  rx_DeleteMsgPart(pAnalyzeLastMessage := pAnalyzeLastMessage, nLen := nFindIndex , nPos := 1);
ELSE
  // end of message detected
  nFindIndex := FIND2(pAnalyzeLastMessage, ADR(');'));
  IF nFindIndex > 0 THEN
    (*Last sector is indicated with '-1'*)
    nSector := STRING_TO_DINT(LEFT(pAnalyzeLastMessage^, (UDINT_TO_INT(nFindIndex) - 1)));
  
    rx_DeleteMsgPart(pAnalyzeLastMessage := pAnalyzeLastMessage, nLen := nFindIndex + 1, nPos := 1);
  END_IF;
END_IF;

rx_ParseHeader := TRUE;
END_METHOD

(*
  Parse a point entry from string.
  And removes this string part from pAnalyzeLastMessage.
  :return: TRUE if point is valid
*)
METHOD PRIVATE rx_ParsePoint : BOOL
VAR_INPUT
  pAnalyzeLastMessage    : POINTER TO STRING(GVL_TcpIp.TCP_RXDATA_SIZE);  // telegram string for analysis
END_VAR
VAR_OUTPUT
  sCamResult             : ST_CameraPoint;
  bLast                  : BOOL;
END_VAR
VAR
  nFindIndex             : UDINT;
END_VAR
(*Index of mark (T)*)
nFindIndex := FIND2(pAnalyzeLastMessage, ADR(','));
IF nFindIndex > 0 THEN
  sCamResult.id := STRING_TO_UDINT(LEFT(pAnalyzeLastMessage^, (UDINT_TO_INT(nFindIndex) - 1)));
  
  rx_DeleteMsgPart(pAnalyzeLastMessage := pAnalyzeLastMessage, nLen := nFindIndex , nPos := 1);
END_IF;

(*rx*)
nFindIndex := FIND2(pAnalyzeLastMessage, ADR(','));
IF nFindIndex > 0 THEN
  sCamResult.x_ref := STRING_TO_DINT(LEFT(pAnalyzeLastMessage^, (UDINT_TO_INT(nFindIndex) - 1)));

  IF    (sCamResult.x_ref < cCameraMinXY)
     OR (sCamResult.x_ref > cCameraMaxXY)
  THEN
    sCamResult.valid := FALSE;
  END_IF;

  rx_DeleteMsgPart(pAnalyzeLastMessage := pAnalyzeLastMessage, nLen := nFindIndex , nPos := 1);
ELSE
  sCamResult.valid := FALSE;
END_IF;
(*ry*)
nFindIndex := FIND2(pAnalyzeLastMessage, ADR(','));
IF nFindIndex > 0 THEN
  sCamResult.y_ref := STRING_TO_DINT(LEFT(pAnalyzeLastMessage^, (UDINT_TO_INT(nFindIndex) - 1)));

  IF    (sCamResult.y_ref < cCameraMinXY)
     OR (sCamResult.y_ref > cCameraMaxXY)
  THEN
    sCamResult.valid := FALSE;
  END_IF;

  rx_DeleteMsgPart(pAnalyzeLastMessage := pAnalyzeLastMessage, nLen := nFindIndex , nPos := 1);
ELSE
  sCamResult.valid := FALSE;
END_IF;

(*lx*)
nFindIndex := FIND2(pAnalyzeLastMessage, ADR(','));
IF nFindIndex > 0 THEN
  sCamResult.lx := STRING_TO_DINT(LEFT(pAnalyzeLastMessage^, (UDINT_TO_INT(nFindIndex) - 1)));

  IF    (sCamResult.lx < cCameraMinXY)
     OR (sCamResult.lx > cCameraMaxXY)
  THEN
    sCamResult.valid := FALSE;
  END_IF;

  rx_DeleteMsgPart(pAnalyzeLastMessage := pAnalyzeLastMessage, nLen := nFindIndex , nPos := 1);
ELSE
  sCamResult.valid := FALSE;
END_IF;
(*ly*)
nFindIndex := FIND2(pAnalyzeLastMessage, ADR(','));
IF nFindIndex > 0 THEN
  sCamResult.ly := STRING_TO_DINT(LEFT(pAnalyzeLastMessage^, (UDINT_TO_INT(nFindIndex) - 1)));

  IF    (sCamResult.ly < cCameraMinXY)
     OR (sCamResult.ly > cCameraMaxXY)
  THEN
    sCamResult.valid := FALSE;
  END_IF;

  rx_DeleteMsgPart(pAnalyzeLastMessage := pAnalyzeLastMessage, nLen := nFindIndex , nPos := 1);
ELSE
  sCamResult.valid := FALSE;
END_IF;

(*v*)
nFindIndex := FIND2(pAnalyzeLastMessage, ADR(','));
IF nFindIndex > 0 THEN
  IF STRING_TO_INT(LEFT(pAnalyzeLastMessage^, (UDINT_TO_INT(nFindIndex) - 1))) = 1 THEN
    sCamResult.valid := TRUE;
  ELSE
    sCamResult.valid := FALSE;
  END_IF;

  rx_DeleteMsgPart(pAnalyzeLastMessage := pAnalyzeLastMessage, nLen := nFindIndex , nPos := 1);
ELSE
  sCamResult.valid := FALSE;
END_IF;
(*x*)
nFindIndex := FIND2(pAnalyzeLastMessage, ADR(','));
IF nFindIndex > 0 THEN
  sCamResult.x := STRING_TO_DINT(LEFT(pAnalyzeLastMessage^, (UDINT_TO_INT(nFindIndex) - 1)));

  IF    (sCamResult.x < cCameraMinXY)
     OR (sCamResult.x > cCameraMaxXY)
  THEN
    sCamResult.valid := FALSE;
  END_IF;

  rx_DeleteMsgPart(pAnalyzeLastMessage := pAnalyzeLastMessage, nLen := nFindIndex , nPos := 1);
ELSE
  sCamResult.valid := FALSE;
END_IF;
(*y*)
nFindIndex := FIND2(pAnalyzeLastMessage, ADR(','));
IF (nFindIndex > 0) AND (nFindIndex <= 8) THEN  (*nFindIndex is > 8 if a second message is in the frame*)
  sCamResult.y := STRING_TO_DINT(LEFT(pAnalyzeLastMessage^, (UDINT_TO_INT(nFindIndex) - 1)));

  IF    (sCamResult.y < cCameraMinXY)
     OR (sCamResult.y > cCameraMaxXY)
  THEN
    sCamResult.valid := FALSE;
  END_IF;

  rx_DeleteMsgPart(pAnalyzeLastMessage := pAnalyzeLastMessage, nLen := nFindIndex , nPos := 1);
ELSE
  nFindIndex := FIND2(pAnalyzeLastMessage, ADR(');'));
  IF nFindIndex > 0 THEN
    sCamResult.y := STRING_TO_DINT(LEFT(pAnalyzeLastMessage^, (UDINT_TO_INT(nFindIndex) - 1)));
    bLast := TRUE;
    IF    (sCamResult.y < cCameraMinXY)
       OR (sCamResult.y > cCameraMaxXY)
    THEN
      sCamResult.valid := FALSE;
    END_IF;

    rx_DeleteMsgPart(pAnalyzeLastMessage := pAnalyzeLastMessage, nLen := nFindIndex + 1, nPos := 1);
  ELSE
    sCamResult.valid := FALSE;
  END_IF;
END_IF;

rx_ParsePoint := sCamResult.valid;
END_METHOD

(*
  Parse rx test telegrams.
  :return: TRUE if it was a known test telegram, FALSE if other.
*)
METHOD PRIVATE rx_TestMsg : BOOL
VAR_INPUT
  pMessage    : POINTER TO STRING(GVL_TcpIp.TCP_RXDATA_SIZE);   // tcp message string pointer 
END_VAR
VAR
  nFIdx : UDINT;    // string find index
  nFrmIdx : UDINT;
  tDiff : LREAL;
  sTestMsg : T_MaxString;
END_VAR
// rx timestamp
_tTimeRx := F_GetCurDcTaskTime64();

// parse message type
nFIdx := FIND2(pMessage, ADR(sQvTest_Header));
IF nFIdx > 0 THEN  
  IF _bVerbose THEN
    LogLvl(Lvl:=E_LogSeverity.Debug, Msg:=F_Concat2('test_rx: msg received: ', pMessage^));
  END_IF
  
  // test telegram received
  DELETE2( pSrcString := pMessage
         , pDstString := ADR(sTestMsg)
         , nDstSize   := SIZEOF(sTestMsg)
         , nLen       := (nFIdx + INT_TO_UDINT(LEN(sQvTest_Header)) - 1)
         , nPos       := 1);

  // strip QR start and end characters
  FindAndDeleteChar(pSrcString:=ADR(sTestMsg), pDstString:=ADR(sTestMsg), nDstSize:=SIZEOF(sTestMsg), sDeleteChar:='<');
  FindAndDeleteChar(pSrcString:=ADR(sTestMsg), pDstString:=ADR(sTestMsg), nDstSize:=SIZEOF(sTestMsg), sDeleteChar:=';');
  
  // Parse per test message type, e.g.  <QR_CI_1;
  // -- qv input frame timing test
  IF sQvTest_CI = LEFT(sTestMsg, LEN(sQvTest_CI)) THEN
    // strip header and test indication
    DELETE2( pSrcString := ADR(sTestMsg)
           , pDstString := ADR(sTestMsg)
           , nDstSize   := SIZEOF(sTestMsg)
           , nLen       := (1 + INT_TO_UDINT(LEN(sQvTest_CI)) - 1)
           , nPos       := 1);
    // frame number
    nFrmIdx := TO_UINT(sTestMsg);
    IF nFrmIdx <= nC_MaxRxTimingEntries THEN
      _tTimeFrames_TestMsg[nFrmIdx] := F_GetCurDcTaskTime64();     // save test input frame timestamp
      _tTimeFramesMs_TestMsg[nFrmIdx] := TO_LREAL((_tTimeFrames_TestMsg[nFrmIdx]-_tTimeTrigger)/EC_DCTIME_TICKSPERMSEC64);
    END_IF
    rx_TestMsg := TRUE;
    
  // -- qv loop time test frame response
  ELSIF sQvTest_Loop = LEFT(sTestMsg, LEN(sQvTest_Loop)) THEN
    tDiff := TO_LREAL((_tTimeRx - _tTimeTx) / EC_DCTIME_TICKSPERMSEC64); // calc time elapsed in [ms]
    _sTimeElapsed := F_Concat2(TO_STRING(tDiff),'ms');
    LogLvl(Lvl:=E_LogSeverity.Debug, Msg:=F_Concat2('rx_test: Loop time=', _sTimeElapsed));
    rx_TestMsg := TRUE;
  
  // -- unknown test message
  ELSE
    ;
	END_IF
ELSE
  ; // other telegram
END_IF
END_METHOD

METHOD PRIVATE saveAuswertungPoint : ST_DeformationPointAccurate
VAR_INPUT
  sCamPoint : ST_CameraPoint;
END_VAR
VAR_OUTPUT
  bOK : BOOL;   // conversion has been done correctly (ok as well if point is invalid!)
END_VAR
VAR
  nMarkIndex        : UDINT;
  fDistortionFactor : LREAL;                 (*distortion factor*)
END_VAR
(*convert and save Auswertungs point*)
IF NOT getPointIndex(nId:=sCamPoint.id, nIndex=>nMarkIndex) THEN
  LogError(F_Concat3('Auswertung point with Id: ', TO_STRING(sCamPoint.id), ' not found, ignore'));
  bOK := FALSE;
  RETURN;
END_IF

(*----- calculate print point position -----*)
(*Actual position of distinctive mark*)
(*NOTE: camera points have a different resolution! camera 300dpi * 16=4800dpi*)
IF sTeachPoints[nMarkIndex].x_teach_Print = 0 THEN 
  (*Fully automatic mode*)
  sTeachPoints[nMarkIndex].x_Print := FC_CONV_SUBPX_TO_M( sCamPoint.y
                                                          , LREAL_TO_UDINT(cCameraResolution)
                                                          , LREAL_TO_UDINT(cCameraResolutionSubpixel)) * 1000;  (*[m] => [mm]*)
ELSE
  (*Semi automatic mode*)
  sTeachPoints[nMarkIndex].x_Print :=     sTeachPoints[nMarkIndex].x_ref_Print
                                        + sTeachPoints[nMarkIndex].x_teach_Print
                                        - FC_CONV_SUBPX_TO_M( sCamPoint.y
                                                            , LREAL_TO_UDINT(cCameraResolution)
                                                            , LREAL_TO_UDINT(cCameraResolutionSubpixel)) * 1000;  (*[m] => [mm]*)
END_IF;
IF sTeachPoints[nMarkIndex].y_teach_Print = 0 THEN 
  (*Fully automatic mode*)
  sTeachPoints[nMarkIndex].y_Print :=   ((fPrintUnitWidthTAct/2 + fCameraWidthTC/2) * 1000)  (*[m] => [mm]*)
                                        - (  DINT_TO_LREAL(sCamPoint.x)
                                           / (fCameraRealResolution * cCameraResolutionSubpixel) * 25.4);  (*[mm]*)
ELSE
  (*Semi automatic mode*)
  sTeachPoints[nMarkIndex].y_Print :=     sTeachPoints[nMarkIndex].y_ref_Print
                                        + sTeachPoints[nMarkIndex].y_teach_Print
                                        - (  DINT_TO_LREAL(sCamPoint.x)
                                           / (fCameraRealResolution * cCameraResolutionSubpixel) * 25.4);  (*[mm]*)
END_IF;

// save cam point for visu
sCameraPoints[nMarkIndex] := sCamPoint;

(*----- create cam correction point -----*)
(*NOTE: correction will be rounded to [px]*)
saveAuswertungPoint.x_ref := F_MeterToSubPixelReal( sTeachPoints[nMarkIndex].x_ref_Print * 0.001      (*[mm] => [m]*)
                                     , UDINT_TO_LREAL(_nPrintUnitResolution));             (*Result should be in pixels*)                           
saveAuswertungPoint.y_ref := F_MeterToSubPixelReal( sTeachPoints[nMarkIndex].y_ref_Print * 0.001      (*[mm] => [m]*)
                                     , UDINT_TO_LREAL(_nPrintUnitResolution));             (*Result should be in pixels*)       
fCameraDelay := F_SubPixelToMeter(lPosSubPx:=_nCamStartPosDeviation, fResSubPx:=UDINT_TO_LREAL(_nPrintUnitResolution*_nPrintUnitSubPx));
saveAuswertungPoint.dx    := F_MeterToSubPixelReal( (sTeachPoints[nMarkIndex].x_ref_Print - sTeachPoints[nMarkIndex].x_Print) * 0.001  (*[mm] => [m]*)
                                     + fCameraDelay                                        (*apply camera trigger jitter*)
                                     , UDINT_TO_LREAL(_nPrintUnitResolution));             (*Result should be in pixels*)
                                     
(*Distortion due to expansion of print unit, calculate factor*)
fDistortionFactor := ((_fPrintUnitWidthTC / 2 * 1000) - sTeachPoints[nMarkIndex].y_ref_Print) / (_fPrintUnitWidthTC / 2 * 1000);
saveAuswertungPoint.dy := F_MeterToSubPixelReal( (  (sTeachPoints[nMarkIndex].y_ref_Print - sTeachPoints[nMarkIndex].y_Print)
                                     + fCameraAdjustmentY
                                     + ((fPrintUnitWidthDiff * 1000 / 2) * fDistortionFactor)   (*Distortion due to expansion of print unit*)
                                     + (fPrintUnitCenterOffsetTAct - fCameraCenterOffsetTAct)   (*Compensation due to unilateral expansion*)
                                    ) * 0.001  (*[mm] => [m]*)
                                  , UDINT_TO_LREAL(_nPrintUnitResolution));             (*Result should be in pixels*)
                                  
// not used entries
saveAuswertungPoint.index := 0; // optional: TO_DINT(sCamPoint.id);
saveAuswertungPoint.col := 0;
saveAuswertungPoint.row := 0;
saveAuswertungPoint.valid := sCamPoint.valid;
IF NOT sCamPoint.valid THEN     // erase spurious corrections on invalid points
  saveAuswertungPoint.dx := 0;
  saveAuswertungPoint.dy := 0;
END_IF
nNbMarksScanned := nNbMarksScanned + 1;
bOK := TRUE;
END_METHOD

METHOD PRIVATE saveTeachPoint
VAR_INPUT
  sCamPoint : ST_CameraPoint;
END_VAR
(*save teach point in table*)
// NOTE: mark ID unique and does not match the array index! 
IF nNbMarksTeach = GVL_Camera.cMaxNbMarks THEN 
  LogLvl(Lvl:=E_LogSeverity.Error, Msg:=F_Concat4('Too many marks received max. allowed: ', TO_STRING(GVL_Camera.cMaxNbMarks), ' ignore mark with id:', TO_STRING(sCamPoint.id)));
  RETURN;
END_IF

// save next teach mark
nNbMarksTeach := nNbMarksTeach + 1;
sCameraPoints[nNbMarksTeach] := sCamPoint;
END_METHOD

(*
  Set mode to camera.
  :return: TRUE if success
*)
METHOD setCameraMode : BOOL
VAR_INPUT
  eCameraMode : E_CameraMode;
END_VAR
IF eCameraMode = E_CameraMode.XYR OR   // supported modi
   eCameraMode = E_CameraMode.Auto OR
   eCameraMode = E_CameraMode.Live OR 
   eCameraMode = E_CameraMode.Trend THEN
   
  _eCameraMode := eCameraMode;  // set desired mode
  setCameraMode := TRUE;
ELSE
  LogError(F_Concat3('Camera mode=', TO_STRING(eCameraMode), ' not supported by camera'));
  _eCameraMode := E_CameraMode.NoCorrection;
END_IF
END_METHOD

METHOD SimEnter : BOOL
VAR_INST
  sSimMsg         : CalmarCompTcpIp.ST_TcpMsg;
  nFrameSize      : UDINT := 2048;
  nMarksPerFrame  : UDINT := 4;
END_VAR
IF NOT bSimEnable THEN RETURN; END_IF

IF    _nSimMode = 0 THEN
   //nNbMarksTeach := 4; // just somebigger than 2
   //nNbMarks := nNbMarksTeach;
ELSIF _nSimMode = 1 THEN
  // use external camera simulation script
  nFrameNr := 0;
ELSIF _nSimMode = 2 THEN
  // send directly some messages
  sSimMsg.stRemoteAddr.sAddr:='127.0.0.1';
  sSimMsg.stRemoteAddr.nPort:=3000;
  //v100 teach
  //rx_callback(sMessage:='<position(100,T,39,3,125,0,0,0,0,1,7184,7184,126,0,0,0,0,1,7184,26080,127,0,0,0,0,1,7184,35520,128,0,0,0,0,1,7184,54416,129,0,0,0,0,1,7168,73312,130,0,0,0,0,1,7184,82768,131,0,0,0,0,1,7184,101664,132,0,0,0,0,1,7184,120560,133,0,0,0,0,1,7184,139456,134,0,0,0,0,1,7184,148912,135,0,0,0,0,1,7184,167808,136,0,0,0,0,1,7168,186704,137,0,0,0,0,1,63872,7184,138,0,0,0,0,1,63872,26080,139,0,0,0,0,1,63872,35520,140,0,0,0,0,1,63872,54416,141,0,0,0,0,1,63872,73312,142,0,0,0,0,1,63872,82768,143,0,0,0,0,1,63872,101664,144,0,0,0,0,1,63872,120560,145,0,0,0,0,1,63872,139456,146,0,0,0,0,1,63872,148912,147,0,0,0,0,1,63872,167808,148,0,0,0,0,1,63872,186704,149,0,0,0,0,1,130016,7168,150,0,0,0,0,1,130016,26080,151,0,0,0,0,1,130016,35520,152,0,0,0,0,1,130016,54416,153,0,0,0,0,1,130016,73312,154,0,0,0,0,1,130016,82768,155,0,0,0,0,1,130016,101664,156,0,0,0,0,1,130016,120560,157,0,0,0,0,1,130016,139456,158,0,0,0,0,1,130016,148912,159,0,0,0,0,1,130016,167808,160,0,0,0,0,1,130016,186704,161,0,0,0,0,1,35520,7168,162,0,0,0,0,1,35520,5441);');
  //v110 teach
  sSimMsg.sMessage:= '<position(110,T,38,12,1,0,0,0,0,1,7184,7184,2,0,0,0,0,1,7184,26080,4,0,0,0,0,1,7184,35520,128,0,0,0,0,1,7184,54416,5,0,0,0,0,1,7168,73312,130,0,0,0,0,1,7184,82768,131,0,0,0,0,1,7184,101664,132,0,0,0,0,1,7184,120560,133,0,0,0,0,1,7184,139456,134,0,0,0,0,1,7184,148912,135,0,0,0,0,1,7184,167808,136,0,0,0,0,1,7168,186704,137,0,0,0,0,1,63872,7184,138,0,0,0,0,1,63872,26080,139,0,0,0,0,1,63872,35520,140,0,0,0,0,1,63872,54416,141,0,0,0,0,1,63872,73312,142,0,0,0,0,1,63872,82768,143,0,0,0,0,1,63872,101664,144,0,0,0,0,1,63872,120560,145,0,0,0,0,1,63872,139456,146,0,0,0,0,1,63872,148912,147,0,0,0,0,1,63872,167808,148,0,0,0,0,1,63872,186704,149,0,0,0,0,1,130016,7168,150,0,0,0,0,1,130016,26080,151,0,0,0,0,1,130016,35520,152,0,0,0,0,1,130016,54416,153,0,0,0,0,1,130016,73312,154,0,0,0,0,1,130016,82768,155,0,0,0,0,1,130016,101664,156,0,0,0,0,1,130016,120560,157,0,0,0,0,1,130016,139456,158,0,0,0,0,1,130016,148912,159,0,0,0,0,1,130016,167808,160,0,0,0,0,1,130016,186704,161,0,0,0,0,1,35520,7168,162,0,0,0,0,1,35520,5441);';
  //points 1 to 38
  //sSimMsg.sMessage:= '<position(110,T,38,12,1,0,0,0,0,1,7184,7184,2,0,0,0,0,1,7184,26080,3,0,0,0,0,1,7184,35520,4,0,0,0,0,1,7184,54416,5,0,0,0,0,1,7168,73312,6,0,0,0,0,1,7184,82768,7,0,0,0,0,1,7184,101664,8,0,0,0,0,1,7184,120560,9,0,0,0,0,1,7184,139456,10,0,0,0,0,1,7184,148912,11,0,0,0,0,1,7184,167808,12,0,0,0,0,1,7168,186704,13,0,0,0,0,1,63872,7184,14,0,0,0,0,1,63872,26080,15,0,0,0,0,1,63872,35520,16,0,0,0,0,1,63872,54416,17,0,0,0,0,1,63872,73312,18,0,0,0,0,1,63872,82768,19,0,0,0,0,1,63872,101664,20,0,0,0,0,1,63872,120560,21,0,0,0,0,1,63872,139456,22,0,0,0,0,1,63872,148912,23,0,0,0,0,1,63872,167808,24,0,0,0,0,1,63872,186704,25,0,0,0,0,1,130016,7168,26,0,0,0,0,1,130016,26080,27,0,0,0,0,1,130016,35520,28,0,0,0,0,1,130016,54416,29,0,0,0,0,1,130016,73312,30,0,0,0,0,1,130016,82768,31,0,0,0,0,1,130016,101664,32,0,0,0,0,1,130016,120560,33,0,0,0,0,1,130016,139456,34,0,0,0,0,1,130016,148912,35,0,0,0,0,1,130016,167808,36,0,0,0,0,1,130016,186704,37,0,0,0,0,1,35520,7168,38,0,0,0,0,1,35520,5441);';
  rx_callback(sMessage:=sSimMsg);
END_IF
END_METHOD

METHOD SimExit : BOOL
IF NOT bSimEnable THEN RETURN; END_IF

IF    _nSimMode = 0 THEN
  ;  // no action
ELSIF _nSimMode = 1 THEN
  nFrameNr := 0;
ELSIF _nSimMode = 2 THEN
  ;  // no action
END_IF
END_METHOD

(*
  External camera simulation script. 
  Simulates the line camera. Opens a TcpIp server where the the linecam plc client can conect to...
*)
METHOD SimulateCamera
VAR_INST
  rfTrig_En : RF_TRIG;
  tOnFrame  : TON;
END_VAR
VAR
  ams_host : STRING;
  ams_port : UINT;
  cmd : STRING;
  
  tFrameTime : TIME;
END_VAR
IF _nSimMode <> 1 THEN RETURN; END_IF   // only cam simulation

// simulation enable / disable
rfTrig_En(CLK:=_bSimulate);
IF rfTrig_En.RT THEN 
  // --- start simulation -----
  LogLvl(Lvl:=E_LogSeverity.Debug, Msg:='Start CamSimulation');

  fbScriptCamSim.Init(sScriptDir:=F_Concat2(_aCamSimScriptPath, 'Tools\CameraTest\'));
  fbScriptCamSim.sStartScriptName := 'Start.bat';
  (* Script parameter:
    parser.add_argument("ams_host", help="AmsNetId of host system")
    parser.add_argument("ams_port", help="AmsPort of host system", type=int)
    parser.add_argument("plc_path", help="plc interface (base) path")
    parser.add_argument("cam_ip", help="camera ip address")
    parser.add_argument("cam_port", help="camera port")
    parser.add_argument("--sim_mode", help="simulation enabled", type=bool)
  *)
  // build cmd line string dynamically 
  ams_host := '';
  ams_port := TwinCAT_SystemInfoVarList._AppInfo.AdsPort; 
  cmd := F_Concat7(ams_host,' ',TO_STRING(ams_port),' ',THIS^.InstanceName,' ',F_Concat3('127.0.0.1',' ',TO_STRING(5030)));
  fbScriptCamSim.Start(cmd);
  
ELSIF rfTrig_En.FT THEN 
  // --- stop/exit simulation ------
  LogLvl(Lvl:=E_LogSeverity.Debug, Msg:='Stop CamSimulation');
  // stop script
  fbScriptCamSim.Stop(nPID := THIS^.nScriptPID);
END_IF

// --- run script command ------
IF NOT fbScriptCamSim.bBusy THEN 
  IF fbScriptCamSim.bError THEN //Launch error
    LogError(F_Concat2('Script error=', TO_STRING(fbScriptCamSim.nErrId)));
  ELSE //Launch done
    ;
  END_IF
END_IF

// --- script live interface -------
IF _bCamTriggerStarted THEN
  IF tOnFrame.Q THEN
    nFrameNr := nFrameNr + 1; // demand next frame
	END_IF
  tFrameTime := REAL_TO_TIME(((84.6667 / 1_000_000) * 0.5)*1000*1024);  // 1024px @300dpi with speed 0.5m/s
  tOnFrame(IN:=NOT tOnFrame.Q, PT:=tFrameTime);
END_IF
END_METHOD

METHOD SimUpdate : BOOL
VAR_INST
  rfTrigCamTrigger : RF_TRIG;
  sSimMsg          : CalmarCompTcpIp.ST_TcpMsg;
END_VAR
// simulation handling
_rfTrigSim(CLK:=_bSimulate);
IF _rfTrigSim.RT THEN    SimEnter();
ELSIF _rfTrigSim.FT THEN SimExit(); END_IF
IF NOT _bSimulate THEN RETURN; END_IF

// we are in simulation mode
// - triggered
rfTrigCamTrigger(CLK:=_bCamTriggerStarted);

IF    _nSimMode = 0 THEN
  // direct points stream of all points in trigger
  IF rfTrigCamTrigger.RT THEN
     CreateSimCamPoints();
     _ePossibleMode := E_CameraMode.Live;
  END_IF
  // stream points
  StreamSimCamPoint();
 
ELSIF _nSimMode = 1 THEN
  // use external camera simulation script
  SimulateCamera();
  
ELSIF _nSimMode = 2 THEN
  IF rfTrigCamTrigger.RT THEN
    // send directly some messages
    sSimMsg.sMessage:='<position(110,A,5,1,125,0,0,0,0,1,12196,9766,137,0,0,0,0,1,69013,9660,149,0,0,0,0,1,135374,9496,161,0,0,0,0,1,40589,9699,163,0,0,0,0,1,116414,9527);';
    rx_callback(sMessage:=sSimMsg);
    sSimMsg.sMessage:='<position(110,A,3,2,126,0,0,0,0,1,11602,28300,138,0,0,0,0,1,68917,28190,150,0,0,0,0,1,136214,27951);';
    // also posible: sSimMsg.sMessage:='<position(110,A,3,2,126,0,0,0,0,1,11602,28300,138,0,0,0,0,1,68917,28190,150,0,0,0,0,1,136214,27951);<position(110,A,0,-1);';
    rx_callback(sMessage:=sSimMsg);
    sSimMsg.sMessage:='<position(110,A,0,-1);';
    rx_callback(sMessage:=sSimMsg);
  END_IF
END_IF


tx_test();
END_METHOD

{attribute 'monitoring':='variable'}
PROPERTY sName : STRING
GET
sName := 'LineCam Base';
END_GET
END_PROPERTY

(*
  Sort sCameraPoints list with ascending [.id] 
*)
METHOD sortPoints
VAR
  i, k : UDINT;
  tmpPoint : ST_CameraPoint;
END_VAR
// sort array (increasing id)
FOR i := 1 TO nNbMarksTeach DO
  FOR k := 1 TO nNbMarksTeach-1 DO
    IF sCameraPoints[k].id > sCameraPoints[k+1].id THEN
      tmpPoint := sCameraPoints[k+1];
      sCameraPoints[k+1] := sCameraPoints[k];
      sCameraPoints[k] := tmpPoint;
    END_IF
	END_FOR
END_FOR
END_METHOD

METHOD PRIVATE StreamSimCamPoint : BOOL
VAR_INPUT
END_VAR
VAR
 tCurrent : T_DCTIME64;
 tElapsed : LREAL;
 tCol : LREAL;
 nCol : UDINT;
 nPointCt : UDINT;
 tFrameFirstDelayFix : LREAL := 50; // deleat to first received frame after trigger
 tFrameTimeJitterMax : LREAL := 30; // max. process time for a camera frame to be received after a simulated scan [ms]
END_VAR
VAR_INST
 fbRand : DRAND;
END_VAR
IF IfSpeed = 0 THEN RETURN; END_IF

fbRand();
tCurrent := F_GetCurDcTaskTime64();             // current time 
tElapsed := TO_LREAL((tCurrent-_tTimeTrigger)   // time elapsed after trigger
                  / EC_DCTIME_TICKSPERMSEC64); 
tCol := F_SubPixelToMeter(                      // time for one column  in [ms] 
                  lPosSubPx:=TO_DINT(_nSimCamFrameDepth), 
                  fResSubPx:=_nPrintUnitResolution) * 1000 / IfSpeed;
tElapsed := tElapsed-tFrameFirstDelayFix-(tFrameTimeJitterMax * fbRand.Num);
IF tElapsed < 0 THEN nCol := 0;
ELSE                 nCol := TO_UDINT(tElapsed / tCol);  // current column number
END_IF

nPointCt := nCol*_nSimCamMarksPerFrame;         // current number of points to be streamed

// stream new points
WHILE nNbMarksScanned < nPointCt AND nNbMarksScanned < nNbMarks DO
  // add to container
  IF _iCameraSink<>0 THEN
    stCamPoint := _sSimCamPoints[nNbMarksScanned+1];
    _iCameraSink.AddCamPoint(stCamPoint);
    // add scanned marks
  END_IF;
  nNbMarksScanned := nNbMarksScanned + 1;
END_WHILE
END_METHOD

METHOD PRIVATE tx_test : BOOL
VAR_INPUT
END_VAR
VAR_INST
  _sTestTxMsg               : T_MaxString;
END_VAR
IF _pFbTcpIpClient = 0 THEN RETURN; END_IF

// sent a test message to QR
IF _bTestTx THEN
  _sTestTxMsg := F_Concat4('<', sQvTest_Header, sQvTest_Loop, ';');
  _tTimeTx := F_GetCurDcTaskTime64();
  _pFbTcpIpClient^.send(sMessage:=_sTestTxMsg);
  LogLvl(Lvl:=E_LogSeverity.Debug, Msg:=F_Concat2('test_tx sent: ', _sTestTxMsg));
  _bTestTx := FALSE;
END_IF
END_METHOD

(*
  Check teach points for validy and quality.
*)
METHOD verifyTeachPoints : BOOL
VAR
  lCtr : UDINT;
END_VAR

IF _fFrameLength <> 0 THEN
  nNumFrames := LIMIT(1, TO_UDINT(FC_LREAL_TO_DINT((fImageLength / _fFrameLength) + 1)), GVL_Camera.cMaxNbSectors); 
END_IF
bNotAllFramesContainTeachPoints := FALSE;
FOR lCtr := 1 TO nNumFrames DO
  IF nNumPointsPerSectorT[lCtr] = 0 THEN
    bNotAllFramesContainTeachPoints := TRUE;
	END_IF
END_FOR


bNotEnoughTeachPoints := FALSE;
IF    nNumPointsPerSectorT[1] < 2  THEN _ePossibleMode := E_CameraMode.NoCorrection; bNotEnoughTeachPoints := TRUE; //< 2 points in first frame
ELSIF nNumPointsPerSectorT[1] <= 2 THEN _ePossibleMode := E_CameraMode.XYR;          bNotEnoughTeachPoints := TRUE; //< 3 points in first frame
ELSE
  _ePossibleMode := E_CameraMode.Live;
END_IF


// teach is valid
_bTeachOk       := TRUE;
END_METHOD

END_FUNCTION_BLOCK

// ---- POUs/Print/Camera/LineCamera/FB_LineCamera106.TcPOU
(*
  QualiVision line camera system
  DMAX106.   
*)
FUNCTION_BLOCK FB_LineCamera106 EXTENDS FB_LineCamera

VAR CONSTANT
  cCameraWidth106           : DINT := 13440;   (*Camera width [px]*)
  cCameraMechOffsetTC106    : REAL :=  88.0;   (*Camera mechanical offset at calibration temp [mm]*)
  cMechOffsetCameraToPU106  : REAL :=  30.31;  (*Camera mechanical offset to PrintUnit [mm]*)
  cPrintUnitMechOffsetTC106 : REAL := 31.4747; (*PrintUnit mechanical offset at calibration temp [mm]*)
END_VAR

SUPER^();

METHOD InitLineCamera
VAR_INPUT
  nPrintUnitResolution         : UDINT;    (*printhead pixel resolution [dpi]*)
  nPrintUnitSubPx              : UDINT;    (*print unit subPixel resolution [SubPx]*)
  nPrintUnitWidth              : UDINT;    (*print unit width in [px]*)
  iCameraTrigger               : I_CameraTrigger;
END_VAR
(*Init for dmax type*)
_nCameraWidth           := cCameraWidth106;
_fCameraMechOffsetTC    := cCameraMechOffsetTC106;
_fMechOffsetCameraToPU  := cMechOffsetCameraToPU106;
_fPrintUnitMechOffsetTC := cPrintUnitMechOffsetTC106;

SUPER^.InitLineCamera( nPrintUnitResolution := nPrintUnitResolution
                      , nPrintUnitSubPx := nPrintUnitSubPx
                      , nPrintUnitWidth := nPrintUnitWidth
                      , iCameraTrigger := iCameraTrigger);
END_METHOD

{attribute 'monitoring':='variable'}
PROPERTY sName : STRING
GET
sName := 'LineCam 106';
END_GET
END_PROPERTY

END_FUNCTION_BLOCK

// ---- POUs/Print/Camera/LineCamera/FB_LineCamera76.TcPOU
(*
  QualiVision line camera system
  DMAX76.   
*)
FUNCTION_BLOCK FB_LineCamera76 EXTENDS FB_LineCamera

VAR CONSTANT
  cCameraWidth76            : DINT :=  9216;   (*Camera width [px]*)
  cCameraMechOffsetTC76     : REAL := 101.5;   (*Camera mechanical offset at calibration temp [mm]*)
  cMechOffsetCameraToPU76   : REAL :=  13.039; (*Camera mechanical offset to PrintUnit [mm]*)
  cPrintUnitMechOffsetTC76  : REAL := 32.9869; (*PrintUnit mechanical offset at calibration temp [mm]*)
END_VAR

SUPER^();

METHOD InitLineCamera
VAR_INPUT
  nPrintUnitResolution         : UDINT;    (*printhead pixel resolution [dpi]*)
  nPrintUnitSubPx              : UDINT;    (*print unit subPixel resolution [SubPx]*)
  nPrintUnitWidth              : UDINT;    (*print unit width in [px]*)
  iCameraTrigger               : I_CameraTrigger;
END_VAR
(*Init for dmax type*)
_nCameraWidth           := cCameraWidth76;
_fCameraMechOffsetTC    := cCameraMechOffsetTC76;
_fMechOffsetCameraToPU  := cMechOffsetCameraToPU76;
_fPrintUnitMechOffsetTC := cPrintUnitMechOffsetTC76;

SUPER^.InitLineCamera( nPrintUnitResolution := nPrintUnitResolution
                      , nPrintUnitSubPx := nPrintUnitSubPx
                      , nPrintUnitWidth := nPrintUnitWidth
                      , iCameraTrigger := iCameraTrigger);
END_METHOD

{attribute 'monitoring':='variable'}
PROPERTY sName : STRING
GET
sName := 'LineCam 76';
END_GET
END_PROPERTY

END_FUNCTION_BLOCK

// ---- POUs/Print/Camera/LineCamera/FB_LineCamera585.TcPOU
(*
  QualiVision line camera system
  DMAX76.   
*)
FUNCTION_BLOCK FB_LineCamera585 EXTENDS FB_LineCamera

VAR CONSTANT
  cCameraWidth585            : DINT := 9216;     (*Camera width [px]*)
  cCameraMechOffsetTC585     : REAL := 101.5;    (*Camera mechanical offset at calibration temp [mm]*)
  cMechOffsetCameraToPU585   : REAL :=  13.039;  (*Camera mechanical offset to PrintUnit [mm]*)
  cPrintUnitMechOffsetTC585  : REAL :=  32.9869; (*PrintUnit mechanical offset at calibration temp [mm]*)
END_VAR

SUPER^();

METHOD InitLineCamera
VAR_INPUT
  nPrintUnitResolution         : UDINT;    (*printhead pixel resolution [dpi]*)
  nPrintUnitSubPx              : UDINT;    (*print unit subPixel resolution [SubPx]*)
  nPrintUnitWidth              : UDINT;    (*print unit width in [px]*)
  iCameraTrigger               : I_CameraTrigger;
END_VAR
(*Init for dmax type*)
_nCameraWidth           := cCameraWidth585;
_fCameraMechOffsetTC    := cCameraMechOffsetTC585;
_fMechOffsetCameraToPU  := cMechOffsetCameraToPU585;
_fPrintUnitMechOffsetTC := cPrintUnitMechOffsetTC585;

SUPER^.InitLineCamera( nPrintUnitResolution := nPrintUnitResolution
                     , nPrintUnitSubPx      := nPrintUnitSubPx
                     , nPrintUnitWidth      := nPrintUnitWidth
                     , iCameraTrigger       := iCameraTrigger
                     );
END_METHOD

{attribute 'monitoring':='variable'}
PROPERTY sName : STRING
GET
sName := 'LineCam 585';
END_GET
END_PROPERTY

END_FUNCTION_BLOCK

// ---- POUs/Print/Camera/MarkCameraWEU/FB_MarkCamera_WEU.TcPOU
(*
  Mark camera system on WEU machine
  1 mark sensor (optional: reverse mode - roll printed in reversed direction, sensor moved to other side)
*)
FUNCTION_BLOCK FB_MarkCamera_WEU EXTENDS FB_CameraBase
VAR_INPUT
  bReadyForPrinting             : BOOL;     // 
  nCurrentPosition              : DINT;     // current print postion
  fCurrentSpeed                 : LREAL;    // current print speed
  bPrintMarkExist               : BOOL;     // [from machine] print mark existing
  bPrintDirReverse              : BOOL;     // [from machine] print substrate in reverse direction
  nUsePerRepeatInLine           : UDINT;    // [from machine] use per repeat
  fMarkSizeDefault              : LREAL;    // mark size "a" [m]
  fMarkDistRepeatToStartMark    : LREAL;    // mark distance from repeat to start mark [m]
  fMarkDistFromCenter           : LREAL;    // mark distance from center [m]
END_VAR
VAR
  fbMarkDefinition   : FB_MarkDefinition;   // mark definition instance (used by MarkDetection)
  fbMarkDetection    : FB_MarkDetection;    // StartPosTrigger, CameraTrigger and MarkDetection (Mark handler for MarkCamera)
  
  // teach info
  _bTeachOk                     : BOOL;
  _nTeachedPoints               : UDINT;
  _nDetectedMarks               : UDINT;
  
  // status
  _bTeachError                  : BOOL;     // teach was not successful
  _bImageLengthError            : BOOL;     // invalid image/repeat length
  _bMarkDefinitionError         : BOOL;     // invalid mark definition
END_VAR
VAR CONSTANT
  fC_MinImageLength : LREAL := 0.05;  // minimal "repeat" length
END_VAR
VAR PERSISTENT
  eMarkMode     : E_MarkMode := E_MarkMode.AutoDefault;   // mark generation/detection mode
  bMarkInverted : BOOL;             // mark triangle are flipped on x axis
  nUsePerRepeat : UDINT := 4;       // number of "use" per repeat
  fMarkSpec_a   : LREAL := 0.005;   // mark spec a [m] - mark width
  fMarkSpec_b   : LREAL := 0.005;   // mark spec b [m] - (optional) triangle length
  fMarkSpec_c   : LREAL := 0.005;   // mark spec c [m] - start mark distance to 0
END_VAR

IF NOT _bInitialized THEN RETURN; END_IF

// The detection work is done in FB_MarkDetection
// This FB just uses(receives) the marks from the external implementation
// - Receives events CamTrigger & CamTriggerDone from MarkDetection
// - Get current marks and send them to the iCameraSink
fbMarkDetection.bSimEnable := _bSimulate;
IF _bSimulate THEN sim_update(); END_IF

fbMarkDetection(
  bEnable:=bReadyForPrinting,
  bAutomaticMode:=TRUE,
  nCurrentPos:=nCurrentPosition,
  fCurrentSpeed:=fCurrentSpeed
);

_bTeachOk := (fbMarkDefinition.nMarks > 0);
_nTeachedPoints := fbMarkDefinition.nMarks;
_nDetectedMarks := fbMarkDefinition.nMarksDetected;

IF nUsePerRepeatInLine <> nUsePerRepeat THEN nUsePerRepeat := nUsePerRepeatInLine; END_IF

IF _bCamTriggerStarted THEN sendCamPoints(); END_IF

fbMarkDefinition.update_view();

METHOD ackErrors
VAR_INPUT
END_VAR
_bTeachError := FALSE;
_bImageLengthError := FALSE;
_bMarkDefinitionError := FALSE;

fbMarkDetection.ackErrors();
END_METHOD

PROPERTY bImageLengthInvalid : BOOL
GET
bImageLengthInvalid := _bImageLengthError;
END_GET
END_PROPERTY

PROPERTY bMarkDetectionErrors : BOOL
GET
bMarkDetectionErrors := fbMarkDetection._bMarkDetectionErrors;
END_GET
END_PROPERTY

PROPERTY bMissingMarks : BOOL
GET
bMissingMarks := fbMarkDetection._bMissingMarks;
END_GET
END_PROPERTY

PROPERTY bTeachError : BOOL
GET
bTeachError := _bTeachError;
END_GET
END_PROPERTY

METHOD CamTriggerDone
IF NOT _bInitialized THEN RETURN; END_IF

// stream lasting points to Worker Camera
IF _bCamTriggerStarted THEN
  sendCamPoints();
  _iCameraSink.fPrintLengthEffective := fbMarkDetection.fEffectiveImageLength;
END_IF

SUPER^.CamTriggerDone();
END_METHOD

{attribute 'monitoring':='call'}
PROPERTY eCameraMode : E_CameraMode
GET
eCameraMode := _eCameraMode;
IF _eCameraMode = E_CameraMode.Auto THEN
  eCameraMode := E_CameraMode.Live;
END_IF
END_GET
END_PROPERTY

PROPERTY eDeviceType : E_CameraDevice
GET
eDeviceType := E_CameraDevice.PrintMark;
END_GET
END_PROPERTY

METHOD GetCamStatus : BOOL
VAR_OUTPUT
  bConnectionOK  : BOOL;    // Camera connected
  bTeachOk       : BOOL;    // Teach successful
  nTeachedPoints : UDINT;   // Teached points for this job
  nScannedPoints : UDINT;   // Scanned points on current sheet
  bCamStarted    : BOOL;    // Camera trigger is active, cam started
  bCamDone       : BOOL;    // Camera finished on last CT
  bErrors        : ARRAY[1..GVL_Camera.nC_NbCamErrors] OF BOOL;  // generic error flag list
END_VAR
bConnectionOK  := TRUE;
bTeachOk       := _bTeachOk;
nTeachedPoints := _nTeachedPoints;
nScannedPoints := _nRxCamPoints;
bCamStarted    := _bCamTriggerStarted;
bCamDone       := _bCamTriggerDone;

GetCamStatus := bConnectionOK AND bTeachOk;   // camera ready
END_METHOD

METHOD InitMarkCamera
VAR_INPUT
  fPrintUnitResolution         : LREAL;    (*printhead pixel resolution [dpi]*)
  fPrintUnitSubPx              : LREAL;    (*print unit subPixel resolution [SubPx]*)
END_VAR
VAR
  bOK : BOOL;
END_VAR
SUPER^.Init( 
  nPrintUnitResolution      := TO_UDINT(fPrintUnitResolution),
  nPrintUnitSubPx           := TO_UDINT(fPrintUnitSubPx), 
  iCameraTrigger            := fbMarkDetection, 
  bUseCameraTrigger         := FALSE, 
  bUseCameraTriggerFeedback := FALSE
);


IF NOT _bInitialized THEN LogError('Init: invalid parameter'); RETURN; END_IF

// -- Mark definition handler
fbMarkDefinition.Init();

// -- Mark detection handler
fbMarkDetection.Init(
  fPrintResolution:=fPrintUnitResolution, 
  fSubPxResolution:=fPrintUnitSubPx, 
  pFbMarkDefinition:=ADR(fbMarkDefinition)
);

_bInitialized := TRUE;
END_METHOD

METHOD mJobStart : BOOL
// parameter checks
IF fImageLength < fC_MinImageLength THEN _bImageLengthError:=TRUE; LogError('JobStart: Repeat length (ImageLength) too small'); END_IF

// mark mode selection based on machine configuration
// No marks => None
// With marks => use AutoDefault or the special mark selected prior in ui
IF NOT bPrintMarkExist THEN 
  LogLvl(Lvl:=E_LogSeverity.Detail, Msg:='JobStart: No Marks exist, use None/Sim mode');
  eMarkMode := E_MarkMode.None;
ELSE
  IF eMarkMode = E_MarkMode.None THEN 
    eMarkMode := E_MarkMode.AutoDefault; 
  END_IF
END_IF

// get mark definition
fMarkSpec_a := fMarkSizeDefault;
fMarkSpec_c := fMarkDistRepeatToStartMark;
//fMarkSpec_b := ;

IF fMarkSpec_a = 0 THEN _bMarkDefinitionError := TRUE; LogError(F_Concat2('JobStart: MarkLength invalid "a"=', TO_STRING(fMarkSpec_a))); END_IF
IF eMarkMode = E_MarkMode.OneTriangle AND fMarkSpec_b = 0 THEN _bMarkDefinitionError := TRUE; LogError(F_Concat2('JobStart: MarkLength invalid "c"=', TO_STRING(fMarkSpec_c))); END_IF

// Teach marks based on job and configuration
IF eCameraMode <> E_CameraMode.NoCorrection THEN
  _bTeachError := NOT fbMarkDefinition.TeachMarks(
    fImageLength:=fImageLength, 
    fImageWidth:=fImageWidth, 
    eMarkMode:=eMarkMode,
    a:=fMarkSpec_a,
    b:=fMarkSpec_b,
    c:=fMarkSpec_c,
    nUses:=nUsePerRepeat,
    bMarkInverted:=bMarkInverted
  );
END_IF
END_METHOD

PROPERTY pFbMarkDefinition : POINTER TO FB_MarkDefinition
GET
pFbMarkDefinition := ADR(fbMarkDefinition);
END_GET
END_PROPERTY

// stream already detected cam points to sink.
METHOD PRIVATE sendCamPoints
VAR
  i : UDINT;
  pMark : POINTER TO ST_MarkDefinition;
END_VAR
WHILE _nRxCamPoints < fbMarkDefinition.nMarksDetected DO
  
  pMark := fbMarkDefinition.getMark(nIdx:=TO_DINT(_nRxCamPoints+1));
  IF pMark <> 0 THEN
    // Send Mark (CamPoint) to CameraSink
    stCamPoint.x_ref := F_MeterToSubPixelReal(  fPosMeter:=pMark^.fPosX                                 (*[m]*)
                                              , fResoSubPx:=UDINT_TO_LREAL(_nPrintUnitResolution));     (*Result should be in pixels*)
    stCamPoint.y_ref := F_MeterToSubPixelReal( fPosMeter:=pMark^.fPosY                                  (*[m]*)
                                              , fResoSubPx:=UDINT_TO_LREAL(_nPrintUnitResolution));     (*Result should be in pixels*)
    stCamPoint.dx    := F_MeterToSubPixelReal( fPosMeter:=pMark^.sState.dx                              (*[m]*)
                                              , fResoSubPx:=UDINT_TO_LREAL(_nPrintUnitResolution));     (*Result should be in pixels*)
    stCamPoint.dy    := F_MeterToSubPixelReal( fPosMeter:=pMark^.sState.dy                              (*[m]*)
                                              , fResoSubPx:=UDINT_TO_LREAL(_nPrintUnitResolution));     (*Result should be in pixels*)
    stCamPoint.valid := pMark^.sState.bSet;
  
    IF _iCameraSink <> 0 THEN
      _iCameraSink.AddCamPoint(sDeformationPoint:=stCamPoint);
    END_IF
  ELSE
    LogWarning(F_Concat2('Requested mark not found, mark Idx=', TO_STRING(_nRxCamPoints+1)));
  END_IF
  
  _nRxCamPoints := _nRxCamPoints + 1;   // next mark
END_WHILE
END_METHOD

(*
  Set mode to camera.
  :return: TRUE if success
*)
METHOD setCameraMode : BOOL
VAR_INPUT
  eCameraMode : E_CameraMode;
END_VAR
IF eCameraMode = E_CameraMode.Auto OR
   eCameraMode = E_CameraMode.NoCorrection OR
   eCameraMode = E_CameraMode.Live
   //eCameraMode = E_CameraMode.Trend 
THEN
   
  _eCameraMode := eCameraMode;  // set desired mode
  setCameraMode := TRUE;
ELSE
  LogError(F_Concat3('Camera mode=', TO_STRING(eCameraMode), ' not supported by camera'));
  _eCameraMode := E_CameraMode.NoCorrection;
END_IF
END_METHOD

METHOD PRIVATE sim_update
// nothing
END_METHOD

{attribute 'monitoring':='variable'}
PROPERTY sName : STRING
GET
sName := 'Printmarks';
END_GET
END_PROPERTY

END_FUNCTION_BLOCK

// ---- POUs/Print/Camera/MarkCameraWEU/FB_MarkDefinition.TcPOU
(*
  Holds Marks definition & current state.
*)
{attribute 'no_explicit_call' := 'do not call this POU directly'} 
FUNCTION_BLOCK FB_MarkDefinition EXTENDS T_NamedBase IMPLEMENTS I_MarkDefinition
VAR
  // marks
  // - mark list
  _nMarks : UDINT;          // number of registered (teached) marks
  sMarkDef : ARRAY[1..200] OF ST_MarkDefinition;   // mark array (teached marks)
  
  // mark states
  _eMarkMode : E_MarkMode;
  _nMarksDetected : UDINT;  // number of detected marks

  // internals
  nMaxMarks : UDINT;
  sLastStartMark : ST_MarkDefinition;       // sampled start mark (because first mark will be overwritten already by next sheet)
  _a : LREAL;               // saved a Size
  
  // View
  _fImageLength, _fImageWidth, _fUseLength, _fDistBetweenMarks : LREAL;
  _nUses, _nMarksPerUse : UDINT;
  _bMarkInverted : BOOL;
  nSelMark : UDINT := 1;
  pSelMark : POINTER TO ST_MarkDefinition;
  bShowDetail : BOOL;
END_VAR
VAR CONSTANT
  // fixed triangle shape definition
  fC_MinUseLength     : LREAL := 0.04;  // minimal "use" length
  fC_MarkLengthMargin : LREAL := 0.1;   // [factor to a langth of mark] for mark length margin (to allow some jitter)
  //view
  nShSzX_px : UDINT := 700;
  nShSzY_px : UDINT := 180;
END_VAR

(*
  Definition of a mark.
  
   SqLength (1/2a or 2a) | TrLength = a -->
   |--------| \
   |        |   \
   |        |     \    -- center --
^  |        |       \
|  |--------|---------
| Height = a

Requirements:
  - StartMark has to be unique (bigger than minimal length of others)
  - Distance between Start and Endmark has to be bigger than length of StartMark + Minimal space
  - Mark has a minimum lenth, so the sensor can see the mark

*)

PROPERTY fMarkLengthMargin : LREAL
GET
fMarkLengthMargin := fC_MarkLengthMargin * _a;
END_GET
END_PROPERTY

(*
  Ge max length of marks.
*)
PROPERTY fMaxMarkLength : LREAL
GET
IF _nMarks > 0 THEN
  fMaxMarkLength := sMarkDef[1].fSqLength + sMarkDef[1].fTrLength;
END_IF
END_GET
END_PROPERTY

(*
  Get minimum length of hte start mark.
*)
PROPERTY fMinMarkLength : LREAL
GET
IF _nMarks > 0 THEN
  fMinMarkLength := sMarkDef[SEL(_nMarks>1, 1, 2)].fSqLength;
END_IF
END_GET
END_PROPERTY

(*
  Get a mark definition.
  nIdx= 1.._nMarks = registered marks
  nIdx= 0 - selects last mark 
  :returns: pointer to mark defintion or 0 if not found
*)
METHOD getMark : POINTER TO ST_MarkDefinition
VAR_INPUT
  nIdx : DINT; // mark index: 1.._nMarks, 0 = last (endMark) 
END_VAR
IF    nIdx = 0 THEN 
  getMark := ADR(sMarkDef[_nMarks]); // last mark (end or last)
ELSIF nIdx > 0 AND nIdx <= TO_DINT(_nMarks) THEN 
  getMark := ADR(sMarkDef[nIdx]);
ELSE 
  LogError(F_Concat2('Invalid mark requested, Idx=', TO_STRING(nIdx)));
END_IF
END_METHOD

METHOD Init : BOOL
VAR_INPUT
END_VAR
nMaxMarks := SIZEOF(sMarkDef) / SIZEOF(sMarkDef[1]);
ResetDefinition();
LogLevel := E_LogSeverity.Info;
END_METHOD

// return TRUE if its a StartMark
METHOD isStartMark : BOOL
VAR_INPUT
  fMarkLength : LREAL;    // mark length in [m]
END_VAR
IF _nMarks > 0 AND_THEN fMarkLength >= sMarkDef[1].fSqLength THEN  // square length of startMark
  isStartMark := TRUE;
END_IF
END_METHOD

(*Number of registered marks*)
PROPERTY nMarks : UDINT
GET
nMarks := _nMarks;
END_GET
END_PROPERTY

(*Number of detected marks*)
PROPERTY nMarksDetected : UDINT
GET
// number of detected marks
nMarksDetected := _nMarksDetected;
END_GET
END_PROPERTY

PROPERTY pLastStartMark : POINTER TO ST_MarkDefinition
GET
pLastStartMark := ADR(sLastStartMark);
END_GET
END_PROPERTY

(*
  Register a mark to camera (teach).
  If mark.nId >= 0 then it will be a detectable mark.
*)
METHOD RegisterMark : BOOL
VAR_INPUT
  sMark : ST_MarkDefinition;
END_VAR
VAR
  pMark : POINTER TO ST_MarkDefinition;
END_VAR
// - for all other teach marks
IF _nMarks >= nMaxMarks THEN LogError('Number of marks exeeded, ignore'); RETURN; END_IF
// we assume first mark is start mark, last mark is end mark (marks need to be registered in sorted order)
// (TODO) otherwise add marks in a sorted way to list
_nMarks := _nMarks + 1;
pMark := ADR(sMarkDef[_nMarks]);
// copy mark data
pMark^ := sMark;

// checks
// - set id if not given
IF pMark^.nId = 0 THEN pMark^.nId := TO_DINT(_nMarks); END_IF
// - start mark requirements
IF _nMarks > 1 THEN   
  // -- start mark length requirement 
  IF pMark^.fSqLength + pMark^.fTrLength >= sMarkDef[1].fSqLength THEN 
    LogError(F_Concat5('RegisterMark: mark not unique, too long: ', TO_STRING(pMark^.fSqLength + pMark^.fTrLength), ' > ', TO_STRING(sMarkDef[1].fSqLength), ' of start min. length'));
  END_IF
END_IF

// view
pMark^.sView.bShow := TRUE;
pMark^.sView.nXPosPx := TO_DINT(nShSzX_px*pMark^.fPosX/SEL(_fImageLength=0, _fImageLength, 1));
pMark^.sView.nYPosPx := TO_DINT(nShSzY_px*pMark^.fPosY/SEL(_fImageWidth=0,  _fImageWidth,  1));
pMark^.sView.colorFill := SEL(pMark^.nId=1, 16#FFAAABB6, 16#FF8E7CC3 );

// clear eventual mark state
MEMSET(destAddr:=ADR(pMark^.sState), 0, SIZEOF(ST_MarkState));

RegisterMark := TRUE;
END_METHOD

METHOD ResetDefinition
VAR
  i : UDINT;
END_VAR
ResetMarkStates();

_nMarks := 0;
_a := 0;

MEMSET(destAddr:=ADR(sMarkDef), fillByte:=0, SIZEOF(sMarkDef));
MEMSET(destAddr:=ADR(sLastStartMark), fillByte:=0, SIZEOF(sLastStartMark));
END_METHOD

(*
  Reset all registered marks
*)
METHOD ResetMarkStates
VAR
  i : UDINT;
END_VAR
// reset detected marks
_nMarksDetected := 0;
// reset mark state only
FOR i:=1 TO _nMarks DO
  MEMSET(destAddr:=ADR(sMarkDef[i].sState), 0, SIZEOF(ST_MarkState));
  sMarkDef[i].sView.colorFill := 16#FFFFFFFF;
END_FOR
//MEMSET(destAddr:=ADR(sLastStartMark.sState), 0, SIZEOF(ST_MarkState));
END_METHOD

METHOD saveMark : BOOL
VAR_INPUT
  pMark : POINTER TO ST_MarkDefinition;
END_VAR
IF pMark = 0 THEN RETURN; END_IF

IF NOT pMark^.sState.bMissed THEN
  pMark^.sView.colorFill := 16#FF7AF096; // (light greeen) 
ELSIF pMark^.sState.bMissed THEN 
  pMark^.sView.colorFill := 16#FFFD0000; // (some red)
END_IF

// sample start mark
IF pMark^.nId = 1 THEN 
  sLastStartMark := pMark^;           // save start mark as backup
  sMarkDef[pMark^.nId] := pMark^;     // save in teached mark table
  _nMarksDetected := _nMarksDetected + 1;
  saveMark := TRUE;

ELSIF pMark^.nId > 1 AND pMark^.nId <= TO_DINT(_nMarks) THEN
  sMarkDef[pMark^.nId] := pMark^;     // save in teached mark table
  _nMarksDetected := _nMarksDetected + 1;
  saveMark := TRUE;  
  
ELSE
  LogError(F_Concat3('saveMark: mark with id=', TO_STRING(pMark^.nId), ' not available'));
END_IF
END_METHOD

(*
  Calculate marks (position, shape) and register to mark definition. 
*)
METHOD PRIVATE TeachAuto : BOOL
VAR_INPUT
  a : LREAL;              // a length [m]
  c : LREAL;              // c start distance [m]
  bInverted : BOOL;       // mark inverted (flipped on x-axis)
END_VAR
VAR
  i : UDINT;
  bErr : BOOL;
  numMarks : UDINT;
  sNewMark : ST_MarkDefinition;
END_VAR

ResetDefinition();

// 
numMarks := _nUses*_nMarksPerUse;
IF numMarks = 0 THEN numMarks := 1; bErr:=TRUE; END_IF   // at least one mark
IF numMarks > 50 THEN numMarks:=50; bErr:=TRUE; LogError('TeachAuto: too many marks, limited to max. internal=50'); END_IF

_fDistBetweenMarks := _fImageLength/numMarks;

// calculate position
FOR i:=1 TO numMarks DO
  sNewMark.fHeight := a;
  sNewMark.fTrLength := a;
  sNewMark.fSqLength := SEL(i>1, 2*a, 0.5*a);
  sNewMark.fPosX := c + (i-1) * _fDistBetweenMarks;
  sNewMark.fPosY := 0;
  sNewMark.bInvertedX := bInverted;
  
  RegisterMark(sMark:=sNewMark);
END_FOR

TeachAuto := NOT bErr;
END_METHOD

(*Setup mark definition, teach marks for job x
  :return: TRUE if OK
*)
METHOD TeachMarks : BOOL
VAR_INPUT
  fImageLength             : LREAL := 1;      // Image length [m]
  fImageWidth              : LREAL := 1;      // Image width [m]
  eMarkMode                : E_MarkMode;      // mode for expected marks
  // mark format
  a       : LREAL;  // a= mark a length [m]
  b       : LREAL;  // b= mark a length [m]
  c       : LREAL;  // c= distance to start mark (from sheet border)
  nUses   : UDINT;  // use per repeat
  bMarkInverted  : BOOL;   // triangles are flipped Y
END_VAR
VAR
  bOk, bErr : BOOL;
END_VAR
_fImageLength := fImageLength;
_fImageWidth := fImageWidth;
_eMarkMode := eMarkMode;
_bMarkInverted := bMarkInverted;
_nUses := nUses;
_fUseLength := _fImageLength/nUses;
_nMarksPerUse := TO_UDINT(FLOOR(_fUseLength/fC_MinUseLength));
_a := a;

bOK := bErr := FALSE;

// checks
IF fImageLength/nUses < fC_MinUseLength THEN bErr:=TRUE; LogError('TeachMarks: Use length too small'); END_IF

// Teach new marks
IF    eMarkMode = E_MarkMode.AutoDefault THEN
  bOk := TeachAuto(a:=a, c:=c, bInverted:=bMarkInverted);
ELSIF eMarkMode = E_MarkMode.OneDefault THEN
  bOk := TeachOneMark(a:=a, c:=c, bInverted:=bMarkInverted);
ELSIF eMarkMode = E_MarkMode.OneTriangle THEN
  bOk := TeachOneTriangle(a:=a, b:=b, c:=c, bInverted:=bMarkInverted);
ELSIF eMarkMode = E_MarkMode.None THEN
  bOk := TeachOneSimMark();
END_IF

TeachMarks := bOk AND NOT bErr;
END_METHOD

(*
  Calculate marks (position, shape) and register to mark definition. 
*)
METHOD PRIVATE TeachOneMark : BOOL
VAR_INPUT
  a : LREAL;    // a length [m]
  c : LREAL;    // c start distance [m]
  bInverted : BOOL;
END_VAR
VAR
  sNewMark : ST_MarkDefinition;
END_VAR

ResetDefinition();

// > default mark (square & triangle)
// calculate position
sNewMark.fHeight := a;
sNewMark.fTrLength := a;
sNewMark.fSqLength := 2 * a;
sNewMark.fPosX := c;
sNewMark.fPosY := 0;
sNewMark.bInvertedX := bInverted;

RegisterMark(sMark:=sNewMark);

TeachOneMark := TRUE;
END_METHOD

(*
  Calculate marks (position, shape) and register to mark definition. 
*)
METHOD PRIVATE TeachOneSimMark : BOOL
VAR_INPUT
END_VAR
VAR
  sNewMark : ST_MarkDefinition;
END_VAR

ResetDefinition();

// > a simulation/generation mark
// calculate position
sNewMark.bVirtual := TRUE;
sNewMark.fHeight := 0.001;
sNewMark.fTrLength := 0.001;
sNewMark.fSqLength := 0;
sNewMark.fPosX := 0;
sNewMark.fPosY := 0;
sNewMark.bInvertedX := FALSE;

RegisterMark(sMark:=sNewMark);

TeachOneSimMark := TRUE;
END_METHOD

(*
  Calculate marks (position, shape) and register to mark definition. 
*)
METHOD PRIVATE TeachOneTriangle : BOOL
VAR_INPUT
  a : LREAL;    // a length [m]
  b : LREAL;    // b length [m]
  c : LREAL;    // c start distance [m]
  bInverted : BOOL;
END_VAR
VAR
  sNewMark : ST_MarkDefinition;
END_VAR

ResetDefinition();

// calculate position
// > triangle only  (squareLen=0)
sNewMark.fHeight := a;
sNewMark.fTrLength := b;
sNewMark.fSqLength := 0;
sNewMark.fPosX := c;
sNewMark.fPosY := 0;
sNewMark.bInvertedX := bInverted;  

RegisterMark(sMark:=sNewMark);

TeachOneTriangle := TRUE;
END_METHOD

METHOD update_view
VAR_INPUT
END_VAR
nSelMark := LIMIT(1, nSelMark, nMaxMarks);
pSelMark := ADR(sMarkDef[nSelMark]);
END_METHOD

END_FUNCTION_BLOCK

// ---- POUs/Print/Camera/MarkCameraWEU/FB_MarkDetection.TcPOU
(*
  Detects Marks and generates StartTrigger based on one EL1252 timestamp input I/O.
  Implements a CameraTrigger instance as well.
  
  Additionally:
    - returns lateral offset (+/- in [m]) to center of detected marks.
    - manages & supervises mark sequence
    - is a CameraTrigger as well
    - supports simulation mode
  
  NOTE: 
    - a mark has always a rising and falling edge of the sensor (triangle)
    - center position is the middle of the triangular mark

*)
FUNCTION_BLOCK FB_MarkDetection EXTENDS T_NamedBase IMPLEMENTS I_StartPosDetect, I_CameraTrigger, I_Sim
VAR_INPUT
  (*EL1252*)
  bIKp_StartSensor          AT%I* : BOOL;             (*Sensor start trigger*)
  tIKp_TimeStampPos         AT%I* : T_DCTIME64;       (*TimeStamp Pos_Edge @EL1252*)
  tIKn_TimeStampNeg         AT%I* : T_DCTIME64;       (*TimeStamp Neg_Edge @EL1252*)

  // configuration
  bEnable                         : BOOL;             (*Enable start pos detection sensor (from extern)*)
  bAutomaticMode                  : BOOL;             (*machine is in automatic mode *)
  nCurrentPos                     : DINT;             (*current position in [SubPx]*)
  fCurrentSpeed                   : LREAL;            (*actual speed of conveyor in [m/s]*)
  bReverse                        : BOOL;             (*reverse printing same roll feeded in opposite direction, check falling edge in this case*)
  
  // Debug & Test
  bManualTrigger                  : BOOL;             // Manual start trigger
  bManualReset                    : BOOL;             // Manaul reset detection
END_VAR
VAR
  bInitOk                         : BOOL;             // fb initialized

  // config
  _fResolution                    : LREAL := 1;       // current used print resolution (dpi*SubPx)
  _pFbMarkDefinition              : POINTER TO FB_MarkDefinition;      // mark definition
  _iCamera                        : I_Camera;         // camera interface
  // settings                                    
  _bUseCameraTrigger              : BOOL;             // (cam specific setting) Generate camera trigger output
  _bUseCameraTriggerFeedback      : BOOL;             // (cam specific setting) Evaluate camera triggered feedback
  _bCamManualTeachMode            : BOOL;             // cam in manual teach mode
  _fImageLength                   : LREAL;            // Image length in [m] configured (should be repeat length)
  _fImageLengthEffective          : LREAL;            // Image length in [m] detected
  _fTriggerDistance               : LREAL;            // Distance between Sensor and Trigger [m]
  _fTriggerLength                 : LREAL := 10;      // Length of trigger signal in ms, min. 3 bus cycles
  _iActiveCam                     : I_CameraTriggerDevice;  // active camera interface (set by Enable() on I_CameraTrigger)

  bCamValid                       : BOOL;             (*camera is valid*)
  bMarksTeached                   : BOOL;             (*definition is valid marks&substrate*)
  bSpeedValid                     : BOOL;             (*speed is valid*)
  bTriggerArmed                   : BOOL;             (*trigger is armed*)
  bDetectionRunning               : BOOL;             (*detection running an initial start mark was found*)
  bSheetActive                    : BOOL;             (*sheet is scanning*)
    
  // helper
  rfT_Enable                      : RF_TRIG;          // edge detection
  bFound                          : BOOL;             // a mark found
  bTypeStartMark                  : BOOL;             // it is type of start mark
  isMarkMissing                   : BOOL;
  nMarkSelection                  : UDINT := 1;       // Current selected mask to search
  pMarkSearch                     : POINTER TO ST_MarkDefinition;

  
  // time calculations
  tNowDc                          : T_DCTIME64;       // Get Current Timestamp (now)
  fCycleTime                      : LREAL;            // Current calculated cycle time [s]
  
  // I_StartPosDetect
  _bStartTrig                     : BOOL;             // Start Trigger Edge
  _nX0                            : DINT;             // X0 Position [SubPx]
  _bValid                         : BOOL;             // valid start trigger
  
  // errors
  nCtrSensorDetectError           : UDINT;            // (global) error counter for senor detect invalid signals
  nCtrIgnoredMarks                : UDINT;            // (global) error counter for ignored marks
  bNoStartMarkDetected            : BOOL;             // (not implemented yet) no start mark detected after x repeats
  bInvalidRepeatLength            : BOOL;             // (not implemented yet) invalid repeat length (StartMarks too close or too far away from each other)
  nInvalidSignalDetectedPerRepeat : UDINT;            // invalid mark signal in repeat (and ignored)
  nInvalidMarkDetectedPerRepeat   : UDINT;            // invalid mark found in repeat (ignored)

  // err signals --> msg
  _bMarkDetectionErrors           : BOOL;             // invalid sensor signal
  _bMissingMarks                  : BOOL;             // some "valid"* marks were ignored
  
  // simulation & debug
  _bSimEnable                     : BOOL;             // simulation mode enabled
  _nSimMode                       : UDINT;            // simulation mode 0=Simulate Marks, 1=Simulate Sensor 
  _bVerbose                       : BOOL;             // verbose mode
  _fSubstrateGap                  : LREAL;            // Gap between two substrates (sheets/repeats) for simulation
  
  // local for checkForMark
  rfEdgeSensor                    : RF_TRIG;          // edge detection start trigger
  bResetDetection                 : BOOL;             // Reset request for checkForMark() internals

  fRealMarkLength                 : LREAL;
  nRealMarkPosition               : DINT;
  nPosRepeatSupervision           : DINT;             // position sample for supervision of missing StartMarks
  nLastGeneratedStartMarkPosition : DINT;
  bMarkStartDetected              : BOOL;             // mark started
  bMarkEndDetected                : BOOL;             // marks end reached
  bInhibitTrigger                 : BOOL;             // inhibit sensor signals, TRUE=inhibit
  nMarginMarkDist                 : DINT;            // margin distance per mark [m] +/-
  nMarginDelayDist                : DINT;            // cycle time based delay distance [m] +
  
  // history 
  // - repeat
  sRepeatHistory : ARRAY[0..nC_HistorySize-1] OF ST_RepeatHistory;   // detection history
  nRepeatCt : UDINT;                 // history entry selector
  // - marks
  sMarkHistory : ARRAY[0..nC_HistorySize-1] OF ST_MarkDefinition;   // history of detected marks
  nMarkHistoryCt : UDINT;            // history entry selector
  // test
  nSim_Mark_Displacement : UINT;
  fSim_Dx_Fix, fSim_Dy_Fix : LREAL;     // simulate some fix deviation of detected marks [m]
END_VAR
VAR PERSISTENT
  bR_TerminateLast                : BOOL;             // Terminate sheet with last defined & detected mark
  nR_SpeedMavFilterSamples        : UINT := 0;        // moving average filter samples = 0 deactivated
END_VAR
VAR CONSTANT
  fC_MinimalSpeed                 : LREAL := 0.010;   // [m/s] speed valid (used for trigger activation)

  fC_MaxSubstrateFactor           : LREAL := 1.1;     // factor which the sheet length can be max. longer
  fC_MinSubstrateFactor           : LREAL := 0.9;     // factor which the sheet length can be smaller
  nC_MaxRepeatsWithoutStart       : LREAL := 3;       // max repeats (theoretical distance) without a detected start trigger before error
  nC_AreaMarkSensorOk             : INT   := 10;      // [%] Area with the correct arrangement of the mark sensor
  nC_HistorySize                  : UDINT := 20;
  fC_JitterDistPerMark            : LREAL := 0.0005;   // [m] deviation allowed per mark (incrementing as more far in sheet we are to allow streches)
END_VAR

// check parameter
IF NOT bInitOk THEN RETURN; END_IF

// General calculations
bSpeedValid   := fCurrentSpeed > fC_MinimalSpeed;                // speed valid (ignore trigger if not moving)
bCamValid     := SEL(_iActiveCam<>0, FALSE, TRUE);               // camera valid (ignore trigger otherwise)
bMarksTeached    := (_fImageLength > 0 AND _pFbMarkDefinition^.nMarks > 0);
tNowDc        := F_GetCurDcTaskTime64();                         // current dc time (most accurate time stamp we have)
fCycleTime    := calcCycleTime(tCurrent:=tNowDc);                // calculate cycle time of this fb
bTriggerArmed :=  bCamValid AND bSpeedValid AND bEnable AND bMarksTeached AND (bAutomaticMode OR _bCamManualTeachMode OR _bSimEnable);   // trigger

IF bCamValid THEN    // (not yet used) save dynamic changable settings
  _fTriggerDistance := _iActiveCam.fTriggerDistance;
  _fTriggerLength   := _iActiveCam.fTriggerPulseLength;
END_IF

_bValid := _bStartTrig := FALSE;    // default values (outputs and properties)

manualTrigger();     // handle manual trigger


// enable & reset
rfT_Enable(CLK:=bTriggerArmed);             // edge detection for detection started
IF rfT_Enable.RT OR rfT_Enable.FT OR bManualReset THEN Reset(); bManualReset:=FALSE; END_IF;   // reset detection and sheet if trigger fails
IF NOT bEnable THEN RETURN; END_IF    // do nothing if not enabled
IF NOT bTriggerArmed THEN RETURN; END_IF




(*Mark search ----------------------------------------------------------------*)
IF nMarkSelection > _pFbMarkDefinition^.nMarks OR nMarkSelection = 0 THEN nMarkSelection := 1; END_IF  // fix invalid selection
pMarkSearch :=  _pFbMarkDefinition^.getMark(nIdx:=TO_DINT(nMarkSelection));

// --- Simulation for testing
IF _bSimEnable AND _nSimMode = 0 THEN   // simulate some marks for testing
  bFound := SimMarks(pMark:=pMarkSearch, bStartMark=>bTypeStartMark);

// --- Generate masks if none are available
ELSIF pMarkSearch^.bVirtual THEN    // generate marks (for NoMark mode)
  bFound := GenMark(pMark:=pMarkSearch, bStartMark=>bTypeStartMark);

// --- Default by IO signal
ELSE
  bFound := searchForMark(   bSensorSignal := bIKp_StartSensor
                           , tSensorRisingEdge := tIKp_TimeStampPos
                           , tSensorFallingEdge := tIKn_TimeStampNeg
                           , nCurrentPos := nCurrentPos
                           , fSpeed := fCurrentSpeed
                           , bInhibit := bInhibitTrigger
                           , fDuration => //
                           , fDetectedMarkLength => fRealMarkLength
                           , nDetectedMarkPosition => nRealMarkPosition
                           , bStartMark => bTypeStartMark
                         );
END_IF


(*Mark handling ----------------------------------------------------------------*)
IF bFound THEN
  
  // verify if correct mark type-> ignore else
  IF nMarkSelection = 1 AND NOT bTypeStartMark THEN  
    // err - search start mark but other valid found
    nCtrIgnoredMarks := nCtrIgnoredMarks + 1;   // ignored
    nInvalidMarkDetectedPerRepeat := nInvalidMarkDetectedPerRepeat + 1;
    IF _bVerbose THEN LogInfo('Start Mark searched but intermediate found -> ignore mark'); END_IF
    
  ELSIF nMarkSelection > 1 AND bTypeStartMark THEN   
    // err - search intermediate but found start mark
    nCtrIgnoredMarks := nCtrIgnoredMarks + 1;   // ignored
    nInvalidMarkDetectedPerRepeat := nInvalidMarkDetectedPerRepeat + 1;
    IF _bVerbose THEN LogInfo('Start Mark found but searched intermediate -> ignore mark'); END_IF
    
  ELSIF nMarkSelection = 1 AND bTypeStartMark THEN
    // ok - start mark   
    IF _pFbMarkDefinition^.nMarks = 1 THEN    // only one mark --> TERMINATE + START
      //IF (nCurrentPos - _nX0) > (_fSubstrateLength * fC_MinSubstrateFactor ) THEN
        SheetStart(pMark:=pMarkSearch);       // start sheet/repeat
        IF bR_TerminateLast THEN SheetStop(nNewX0:=0); END_IF  // TERMINATE already after single mark scanned
    ELSE                                      // more marks --> START + NEXT
      SheetStart(pMark:=pMarkSearch);         // start sheet/repeat
      nMarkSelection := nMarkSelection + 1;   // next mark
    END_IF
    
  ELSIF nMarkSelection > 1 AND NOT bTypeStartMark THEN
    // ok - intermediate mark
    // search and found other --> NEXT (ev. terminate)
    IF _pFbMarkDefinition^.nMarksDetected < _pFbMarkDefinition^.nMarks THEN
      _pFbMarkDefinition^.saveMark(pMark:=pMarkSearch);           // save mark
      SaveToMarkHistory(pMark:=pMarkSearch);                      // Save to mark history
      IF nMarkSelection = _pFbMarkDefinition^.nMarks THEN         // last mark?
        IF bR_TerminateLast THEN SheetStop(nNewX0:=0); END_IF     // stop 
        nMarkSelection := 1;                                      // search start again
      ELSE
        nMarkSelection := SEL(nMarkSelection<_pFbMarkDefinition^.nMarks, 1, nMarkSelection + 1);  // search next
      END_IF
    END_IF
    
  ELSE
    // err = not covered check
    nCtrIgnoredMarks := nCtrIgnoredMarks + 1;
    nInvalidMarkDetectedPerRepeat := nInvalidMarkDetectedPerRepeat + 1;
    IF _bVerbose THEN LogInfo('Case not covered -> ignore mark'); END_IF
  END_IF 

ELSE
  // inhibit control
  nMarginMarkDist  := F_MeterToSubPixel(fPosMeter:=pMarkSearch^.nId * fC_JitterDistPerMark, fResoSubPx:=_fResolution);
  nMarginDelayDist := F_MeterToSubPixel(fPosMeter:=(1*fCurrentSpeed*fCycleTime), fResoSubPx:=_fResolution);
  IF pMarkSearch^.nId = 1 THEN
    bInhibitTrigger := FALSE;  // release inhibit for first mark
  ELSIF (nCurrentPos - getLastX0() - (getMinMarkPosition(pMark:=pMarkSearch) - nMarginMarkDist)) > 0 THEN
    bInhibitTrigger := FALSE;  // release inhibit
  ELSIF (nCurrentPos - getLastX0() - (getMaxMarkPosition(pMark:=pMarkSearch) + nMarginMarkDist + nMarginDelayDist)) > 0 THEN
    bInhibitTrigger := TRUE;   // set inhibit
  ELSE
    bInhibitTrigger := FALSE;  // release inhibit else
  END_IF
  
  // search if intermediate mark was missed -> create a virtual one
  IF pMarkSearch^.nId > 1 AND (nCurrentPos - getLastX0() - getMaxMarkPosition(pMark:=pMarkSearch) - nMarginMarkDist - nMarginDelayDist) > 0 THEN
    setupMark(
      pMark:=pMarkSearch,
      nDetectedPos:=getLastX0()+F_MeterToSubPixel(fPosMeter:=pMarkSearch^.fPosX, fResoSubPx:=_fResolution),
      fRealMarkLength:=pMarkSearch^.fSqLength+pMarkSearch^.fTrLength/2,
      bMissed:=TRUE
    );
    
    IF _pFbMarkDefinition^.nMarksDetected < _pFbMarkDefinition^.nMarks THEN
      _pFbMarkDefinition^.saveMark(pMark:=pMarkSearch);           // save mark
      SaveToMarkHistory(pMark:=pMarkSearch);                      // Save to mark history
      IF nMarkSelection = _pFbMarkDefinition^.nMarks THEN         // last mark?
        IF bR_TerminateLast THEN SheetStop(nNewX0:=0); END_IF     // stop 
        nMarkSelection := 1;                                      // search start again
      ELSE
        nMarkSelection := SEL(nMarkSelection<_pFbMarkDefinition^.nMarks, 1, nMarkSelection + 1);  // search next
      END_IF
    END_IF
    
  END_IF
END_IF


// --- Error Handling
checkForErrors();


// outputs
// _bStartTrig := // set in SheetStart
// _nX0 :=        // set in SheetStart
_bValid := TRUE;

METHOD ackErrors
VAR_INPUT
END_VAR
nCtrSensorDetectError := 0;
nCtrIgnoredMarks := 0;
_bMarkDetectionErrors := FALSE;
_bMissingMarks := FALSE;
END_METHOD

PROPERTY bManualTeach : BOOL
GET
bManualTeach := _bCamManualTeachMode;
END_GET
SET
_bCamManualTeachMode := bManualTeach;
END_SET
END_PROPERTY

{attribute 'monitoring' := 'call'}
(*Simulation is enabled set/get*)
PROPERTY bSimEnable : BOOL
GET
bSimEnable := _bSimEnable;
END_GET
SET
_bSimEnable := bSimEnable;
END_SET
END_PROPERTY

(*
  A new container detected.
  NOTE: a pulse only
*)
PROPERTY bStartTrig : BOOL
GET
bStartTrig := _bStartTrig;
END_GET
END_PROPERTY

(*
  A valid container detected.
*)
PROPERTY bValid : BOOL
GET
bValid := _bValid;
END_GET
END_PROPERTY

// cycle time in [s]
METHOD PRIVATE calcCycleTime : LREAL
VAR_INPUT
  tCurrent : T_DCTIME64;
END_VAR
VAR_INST
  tLastTimeStamp : T_DCTIME64 := 0;
END_VAR
calcCycleTime := (TO_LREAL(tCurrent) - TO_LREAL(tLastTimeStamp)) * 1E-9;
tLastTimeStamp  := tCurrent;  // memory timestamp
END_METHOD

METHOD PRIVATE checkForErrors
VAR_INST
  nCtrSensorDetectError_mem       : UDINT;            // error counter for senor detect invalid signals
  nCtrIgnoredMarks_mem            : UDINT;            // error counter for ignored marks
  tErrorReport                    : TON;              // check if error increases
  nNumChecks                      : UDINT;
END_VAR

IF nCtrIgnoredMarks > 0 OR nCtrSensorDetectError > 0 THEN 
  // run check timer while error exists
  tErrorReport(IN:=TRUE, PT:=T#15S);

ELSE
  nNumChecks := 0; nCtrSensorDetectError_mem := 0; nCtrIgnoredMarks_mem := 0;
  tErrorReport(IN:=FALSE);
END_IF


IF tErrorReport.Q THEN
  // check if errors did increase some marks -> set error
  tErrorReport(IN:=FALSE);  // stop, restart timer
  IF nCtrSensorDetectError > nCtrSensorDetectError_mem + 3 AND nNumChecks>2 THEN _bMarkDetectionErrors := TRUE; END_IF
  IF nCtrIgnoredMarks > nCtrIgnoredMarks_mem + 3           AND nNumChecks>2 THEN _bMissingMarks := TRUE; END_IF  // TODO: improve to allow x missing per repeat
  nCtrSensorDetectError_mem := nCtrSensorDetectError; 
  nCtrIgnoredMarks_mem := nCtrIgnoredMarks;
  nNumChecks := nNumChecks + 1;
END_IF
END_METHOD

METHOD Disable : BOOL
_iActiveCam := 0;
Disable := TRUE;
END_METHOD

METHOD Enable : BOOL
VAR_INPUT
	iCam	                    : I_CameraTriggerDevice;
  bUseCameraTrigger         : BOOL; //Generate camera trigger
  bUseCameraTriggerFeedback : BOOL; //Use feedback as trigger?
END_VAR
IF iCam = 0 THEN
  Enable := FALSE;
  LogError('setCam failed: invalid reference');
ELSE
  _iActiveCam := iCam;
  Enable     := TRUE;

  // save constant settings
  _bUseCameraTrigger := bUseCameraTrigger;
  _bUseCameraTriggerFeedback := bUseCameraTriggerFeedback;
  
  IF _bUseCameraTrigger OR _bUseCameraTriggerFeedback THEN
    LogWarning('Enable: Camera Trigger output/feedback not yet supported');
	END_IF
END_IF;
END_METHOD

PROPERTY fEffectiveImageLength : LREAL
GET
fEffectiveImageLength := _fImageLengthEffective;
END_GET
END_PROPERTY

PROPERTY fSubstrateGap : LREAL
SET
_fSubstrateGap := fSubstrateGap;
END_SET
END_PROPERTY

(*
  Generate detected marks.
*)
METHOD PRIVATE GenMark : BOOL
VAR_INPUT
  pMark : POINTER TO ST_MarkDefinition;
END_VAR
VAR_OUTPUT
  bStartMark : BOOL;
END_VAR
VAR_INST
  bMarkOn : BOOL;
  n : DINT;
  nImageLengthSubPx : DINT;
END_VAR
IF pMark = 0 THEN RETURN; END_IF

nImageLengthSubPx := F_MeterToSubPixel(fPosMeter:=_fImageLength + _fSubstrateGap, fResoSubPx:=_fResolution);
IF nImageLengthSubPx = 0 THEN RETURN; END_IF


IF NOT bMarkOn THEN  // start new mark
  // create rising edge
  IF pMark^.nId = 1 THEN          // a start mark
    // wait for next StartPosition
    IF ABS(nCurrentPos-nLastGeneratedStartMarkPosition) >= nImageLengthSubPx THEN

      // fix bigger gaps than next sheet (always try to start repeats at a multiple of last repeat)
      IF (nCurrentPos - nLastGeneratedStartMarkPosition) / nImageLengthSubPx > 2 THEN
        nLastGeneratedStartMarkPosition := nLastGeneratedStartMarkPosition + ((((nCurrentPos - nLastGeneratedStartMarkPosition) / nImageLengthSubPx) -1) * nImageLengthSubPx);  // correct to one sheet before 
			END_IF 
      
      nLastGeneratedStartMarkPosition := nLastGeneratedStartMarkPosition + nImageLengthSubPx;      // save last repeat position   
      
      pMark^.sState.nPosXReal := nLastGeneratedStartMarkPosition + F_MeterToSubPixel(fPosMeter:=pMark^.fPosX, fResoSubPx:=_fResolution); // mark detected position
      pMark^.sState.fLengthReal := 0;
      pMark^.sState.dx := 0;
      pMark^.sState.dy := 0;
      pMark^.sState.bInArea := TRUE;
      pMark^.sState.bSet := TRUE;
      bMarkOn := TRUE;
    END_IF
	ELSE
    // wait for next mark position
    IF F_SubPixelToMeter(lPosSubPx:=ABS(nCurrentPos - nLastGeneratedStartMarkPosition), fResSubPx:=_fResolution) >= pMark^.fPosX THEN
     
      pMark^.sState.nPosXReal := nLastGeneratedStartMarkPosition + F_MeterToSubPixel(fPosMeter:=pMark^.fPosX, fResoSubPx:=_fResolution); // 
      pMark^.sState.fLengthReal := 0;
      pMark^.sState.dx := 0;
      pMark^.sState.dy := 0;
      pMark^.sState.bInArea := TRUE;
      pMark^.sState.bSet := TRUE;
      bMarkOn := TRUE;
		END_IF
  END_IF
  
ELSE
  // end mark after one dycle
  bMarkOn := FALSE;
  IF pMark^.nId = 1 THEN bStartMark := TRUE; END_IF  
  GenMark := TRUE;      // reset after one cycle active
END_IF
END_METHOD

// calculate the exact detected position
// :returns: the X0 position
METHOD PRIVATE getExactPosition : DINT
VAR_INPUT
  tNow              : T_DCTIME64;    // current system time
  tEdge             : T_DCTIME64;   // detected time
  nPos              : DINT;          // current (encoder) position at the current time
  fSpeed            : LREAL;       // current speed for the timestamped position correction calculation
END_VAR
VAR
  fCurrentTimeStamp : LREAL;
  fSensor_TimeStamp : LREAL;
  nDeltaPosition    : DINT;       // distance [SubPx]
  fDeltaDistance    : LREAL;      // Distance that the substrate moved between the detection and the treatment of the information
END_VAR
IF _bSimEnable THEN // calculation like DMAX for simulation mode
  fDeltaDistance := UINT64_TO_LREAL(UInt64Sub64(ULINT_TO_ULARGE(tNowDc), ULINT_TO_ULARGE(tEdge))) * 1E-9 * fSpeed;
  getExactPosition := nPos - F_MeterToSubPixel(fPosMeter:=fDeltaDistance, fResoSubPx:=_fResolution);
  RETURN; 
END_IF

// Calculate the original position back from timestamp input trigger (compensated)
fCurrentTimeStamp  := (ULINT_TO_LREAL(tNow) - (GVL_WEU.nC_CurrentTimeStampComp * 1_000)) / 1_000_000.0; // [ms]
fSensor_TimeStamp := (ULINT_TO_LREAL(tEdge) - (GVL_WEU.nC_SensorTimeStampComp  * 1_000)) / 1_000_000.0; // [ms]

// Treatment of the information
fDeltaDistance   := (fCurrentTimeStamp - fSensor_TimeStamp) * 0.001 * fSpeed;	      // Distance in pulses that the substrate has traveled between the sensor detection and the PLC treatment
nDeltaPosition := FC_LREAL_TO_DINT(fDeltaDistance * (1 / (0.0254 / _fResolution)));   // 1/1px*)	(* Travel of the substrate between the time of acquisition and the time of treatment
getExactPosition := nPos - nDeltaPosition;	                                          // Position where the sheet has been detected
END_METHOD

(*
  Get X0 from detected start mark
*)
METHOD PRIVATE getLastX0 : DINT
VAR
  pLastStartMark : POINTER TO ST_MarkDefinition;
END_VAR
pLastStartMark := _pFbMarkDefinition^.pLastStartMark;
IF pLastStartMark <> 0 THEN
  getLastX0 := pLastStartMark^.sState.nPosXReal - F_MeterToSubPixel(fPosMeter:=pLastStartMark^.fPosX, fResoSubPx:=_fResolution);
END_IF
END_METHOD

(*
  Calculate effective distance of mark to X0 [m]
*)
METHOD PRIVATE getMarkDistanceEffective : LREAL
VAR_INPUT
  pMark : POINTER TO ST_MarkDefinition;
END_VAR
VAR
  pFirstMark : POINTER TO ST_MarkDefinition;
END_VAR
IF pMark = 0 THEN RETURN; END_IF

IF pMark^.nId = 1 THEN 
  getMarkDistanceEffective := pMark^.fPosX;
ELSE
  pFirstMark := _pFbMarkDefinition^.getMark(nIdx:=1);
  IF pFirstMark <> 0 THEN
    // real distance between this mark and start mark + fPosX of start mark
    getMarkDistanceEffective := pFirstMark^.fPosX + F_SubPixelToMeter(lPosSubPx:=pMark^.sState.nPosXReal - pFirstMark^.sState.nPosXReal, fResSubPx:=_fResolution);
  END_IF
END_IF
END_METHOD

// get max. mark distance from the sheetStart (teached pos + max. size of mark + margin) [SubPx]
METHOD getMaxMarkPosition : DINT
VAR_INPUT
  pMark : POINTER TO ST_MarkDefinition;
END_VAR
IF pMark = 0 THEN RETURN; END_IF

getMaxMarkPosition := F_MeterToSubPixel(fPosMeter:=pMark^.fPosX + pMark^.fSqLength + pMark^.fTrLength + _pFbMarkDefinition^.fMarkLengthMargin, fResoSubPx:=_fResolution);
END_METHOD

// get max. mark distance from the sheetStart (teached + margin) [SubPx]
METHOD getMinMarkPosition : DINT
VAR_INPUT
  pMark : POINTER TO ST_MarkDefinition;
END_VAR
IF pMark = 0 THEN RETURN; END_IF

getMinMarkPosition := F_MeterToSubPixel(fPosMeter:=pMark^.fPosX - _pFbMarkDefinition^.fMarkLengthMargin, fResoSubPx:=_fResolution);
END_METHOD

METHOD Init
VAR_INPUT
  fPrintResolution      : LREAL := 600;         // print(head) resolution in [dpi]
  fSubPxResolution      : LREAL := 32;          // SubPixel resolution [SubPx], resolution factor (fI_PrintResolution*fI_SubPxResolution=>Output resolution)
  pFbMarkDefinition     : POINTER TO FB_MarkDefinition;
END_VAR
VAR
  i : UDINT;
END_VAR
IF fPrintResolution = 0 OR fSubPxResolution = 0 OR pFbMarkDefinition = 0 THEN LogError('Init: invalid parameter'); RETURN; END_IF

_fResolution := fPrintResolution * fSubPxResolution;
_pFbMarkDefinition:= pFbMarkDefinition;

Reset();

bInitOk := TRUE;
END_METHOD

METHOD PRIVATE manualTrigger : BOOL
VAR_INST
  rfTrig_ManuTrigger : RF_TRIG;
END_VAR
rfTrig_ManuTrigger(CLK:=bManualTrigger);

IF rfTrig_ManuTrigger.RT THEN 
  // LogWarning('manualTrigger not yet implemented');
END_IF

manualTrigger := rfTrig_ManuTrigger.RT;
END_METHOD

(*
  Detected start position X0 (absolute) in [SubPx].
*)
PROPERTY nStartPositionX0 : DINT
GET
nStartPositionX0 := _nX0;
END_GET
END_PROPERTY

(*
  Reset internal state and all marks
*)
METHOD Reset
IF NOT bInitOk THEN RETURN; END_IF

_bValid := FALSE;
_bStartTrig := FALSE;
nMarkSelection := 1; // start mark
bDetectionRunning := FALSE;
nPosRepeatSupervision := nCurrentPos;       // sample activated detection position

// reset camera (release if one is selected)
IF bSheetActive THEN
  IF _iActiveCam <> 0 THEN _iActiveCam.CamTriggerDone(); END_IF   // notify an done/abort
END_IF
_pFbMarkDefinition^.ResetMarkStates();  // reset detected marks
bSheetActive := FALSE;
bResetDetection := TRUE;        // reset checkForMark() state machine

// reset errors
nCtrSensorDetectError := 0;
nCtrIgnoredMarks := 0;
bNoStartMarkDetected := FALSE;
bInvalidRepeatLength := FALSE;
nInvalidSignalDetectedPerRepeat := 0;
nInvalidMarkDetectedPerRepeat := 0;
_bMarkDetectionErrors := FALSE;
_bMissingMarks := FALSE;
END_METHOD

METHOD PRIVATE SaveToMarkHistory
VAR_INPUT
  pMark : POINTER TO ST_MarkDefinition;
END_VAR
VAR
  i : UDINT;
END_VAR
FOR i:=0 TO nC_HistorySize-1 DO sMarkHistory[i].sView.colorFill := 16#FFE2DDDB; END_FOR   // clear selection
nMarkHistoryCt := (nMarkHistoryCt + 1) MOD nC_HistorySize;
sMarkHistory[nMarkHistoryCt] := pMark^;
sMarkHistory[nMarkHistoryCt].sView.colorFill := 16#FF90EE90;
END_METHOD

(*
  Poll sensor signal for triggers and create mark info.
  :return: true if a mark was detected
*)
METHOD PRIVATE searchForMark : BOOL
VAR_INPUT
  bSensorSignal : BOOL;
  tSensorRisingEdge : T_DCTIME64;  // [us]
  tSensorFallingEdge : T_DCTIME64; // [us]
  nCurrentPos : DINT;              // [SubPx]
  fSpeed : LREAL;                  // [m/s]
  bInhibit : BOOL;                 // inhibit sensor signal
END_VAR
VAR_OUTPUT
  fDuration : LREAL;
  fDetectedMarkLength : LREAL;  // [m]
  nDetectedMarkPosition : DINT; // [SubPx]
  bStartMark : BOOL;            // is it a start mark?
END_VAR
VAR_INST
  nAbortMarkAfterDist         : DINT;             // max. length to search for mark end before aborting this mark [SubPx]
  tRisingEdge, tFallingEdge   : T_DCTIME64;       // detected edges
  nRisingPos, nFallingPos     : DINT;             // detected [SubPx] pos
  fLengthByTime : LREAL;
  fLengthByPos  : LREAL;
END_VAR
// reset methods internal states
IF bResetDetection THEN bResetDetection := FALSE;
  bMarkStartDetected := FALSE; bMarkEndDetected := FALSE;
END_IF

// simulate sensor
IF _bSimEnable AND _nSimMode = 1 THEN
  SimSensor(bSensorSimulationSignal=>bSensorSignal, tSensorRising=>tSensorRisingEdge, tSensorFalling=>tSensorFallingEdge);
END_IF

// -- TODO: inhibit control if needed


// --- Use sensor
rfEdgeSensor(CLK:=bSensorSignal);   // edge detection
nAbortMarkAfterDist := F_MeterToSubPixel(fPosMeter:=_pFbMarkDefinition^.fMaxMarkLength + _pFbMarkDefinition^.fMarkLengthMargin + fCycleTime*fCurrentSpeed, fResoSubPx:=_fResolution); // mark len + margin + one cycle


// -- rising edge detection
IF rfEdgeSensor.RT AND NOT bInhibit THEN
  tRisingEdge := tSensorRisingEdge;   // sample input
  nRisingPos  := getExactPosition(tNow:=tNowDc, tEdge:=tRisingEdge, nPos:=nCurrentPos, fSpeed:=fCurrentSpeed);   // position where mark was seen
  bMarkStartDetected := TRUE;
END_IF;

// -- falling edge detection
IF rfEdgeSensor.FT AND NOT bInhibit THEN
  // falling edge
  tFallingEdge := tSensorFallingEdge;
  nFallingPos := getExactPosition(tNow:=tNowDc, tEdge:=tFallingEdge, nPos:=nCurrentPos, fSpeed:=fCurrentSpeed);   // position where mark was seen
  IF NOT bMarkStartDetected THEN
    // ignore
    nCtrSensorDetectError := nCtrSensorDetectError + 1;
    nInvalidSignalDetectedPerRepeat := nInvalidSignalDetectedPerRepeat + 1;
    LogLvl(Lvl:=E_LogSeverity.Debug, Msg:='Missing rising trigger edge before falling edge');
    bResetDetection := TRUE;
  ELSE
    // ok                    
    bMarkEndDetected := TRUE; 
  END_IF
END_IF

// - error handling - abort search for falling edge
IF bMarkStartDetected AND (nCurrentPos - nRisingPos) > nAbortMarkAfterDist THEN      // abort after waiting for end
  // Abort - Expected falling edge missed
  nCtrSensorDetectError := nCtrSensorDetectError + 1;
  nInvalidSignalDetectedPerRepeat := nInvalidSignalDetectedPerRepeat + 1;
  LogLvl(Lvl:=E_LogSeverity.Debug, Msg:=F_Concat2('Mark end not given after [SubPx]:', TO_STRING(nAbortMarkAfterDist)));
  bResetDetection := TRUE;   // reset detection logic
END_IF;


// -- mark evaluation 
IF bMarkStartDetected AND bMarkEndDetected THEN
  // mark found
  fDuration := ABS(ULINT_TO_LREAL(tFallingEdge) - ULINT_TO_LREAL(tRisingEdge));		// Calculate how long the signal was ON
  fLengthByTime := fDuration * fCurrentSpeed * 0.000_000_001;
  fLengthByPos := F_SubPixelToMeter(lPosSubPx:=nFallingPos - nRisingPos, fResSubPx:=_fResolution);
  fDetectedMarkLength := fLengthByPos;
  nDetectedMarkPosition := nRisingPos; // SEL(bReverse, nRisingPos, nFallingPos);
  
  // check if valid
  // - check if mark length is within defined range
  IF fDetectedMarkLength >= (_pFbMarkDefinition^.fMinMarkLength - _pFbMarkDefinition^.fMarkLengthMargin) AND 
     fDetectedMarkLength <= (_pFbMarkDefinition^.fMaxMarkLength + _pFbMarkDefinition^.fMarkLengthMargin) 
  THEN
    // valid
    // - is a startMark type?
    bStartMark := _pFbMarkDefinition^.isStartMark(fMarkLength:=fDetectedMarkLength);
    
    // setup & apply all data to mark structure
    setupMark(
      pMark:=pMarkSearch,
      nDetectedPos:=nDetectedMarkPosition,
      fRealMarkLength:=fDetectedMarkLength,
      bMissed:=FALSE
    );
          
    IF _bVerbose THEN LogInfo(F_Concat4('found ', SEL(bTypeStartMark,'Intermediate','StartMark'), ' ', strMark(pMark:=pMarkSearch))); END_IF
        
    searchForMark := TRUE;              // a valid mark detected
  ELSE 
    // error
    nCtrSensorDetectError := nCtrSensorDetectError + 1;
    nInvalidSignalDetectedPerRepeat := nInvalidSignalDetectedPerRepeat + 1;
    IF _bVerbose THEN LogInfo('Invalid mark lenght found while searching - ignore mark'); END_IF
	END_IF
  
  bResetDetection := TRUE;   // reset detection logic
END_IF
END_METHOD

METHOD SetSubstrateLength
VAR_INPUT
  fSubstrateLength : LREAL;
END_VAR
IF NOT bInitOk THEN RETURN;END_IF;

(*reduced by margin (for endless mode with potential smaller printed repetition)*)
_fImageLength := fSubstrateLength;
END_METHOD

(*
  Setup a detected mark with its details and calculation.
  :returns:  TRUE if valid mark
*)
METHOD PRIVATE setupMark : BOOL
VAR_INPUT
  pMark           : POINTER TO ST_MarkDefinition;     // mark to search for
  nDetectedPos    : DINT;                             // detected position [SubPx]
  fRealMarkLength : LREAL;                            // real detected mark length [m]
  bMissed         : BOOL;                             // missing mark (but generated)
END_VAR
IF pMark = 0 THEN RETURN; END_IF

// apply mark status information
pMark^.sState.bSet := TRUE;
pMark^.sState.bMissed := bMissed;
pMark^.sState.nPosXReal := nDetectedPos;          // save detected mark pos (rising in normal, falling in reverse print)
pMark^.sState.fLengthReal := fRealMarkLength;     // apply detected mark length

// - dx  (based on sheet begin) dx = current mark position - teached mark position ()
pMark^.sState.dx := getMarkDistanceEffective(pMark:=pMark) - pMark^.fPosX;
// - dy  lateral displacement. fHeight/2 (middle) is assumed to be the normal position, the displacement is calculated to this center
pMark^.sState.dy := ((pMark^.sState.fLengthReal - pMark^.fSqLength)/pMark^.fTrLength)*pMark^.fHeight-(pMark^.fHeight/2);

// use (overwrite) with some simulation values
IF    nSim_Mark_Displacement = 1 THEN pMark^.sState.dx := fSim_Dx_Fix; pMark^.sState.dy := fSim_Dy_Fix; 
ELSIF nSim_Mark_Displacement = 2 THEN pMark^.sState.dx := fSim_Dx_Fix * pMark^.nId; pMark^.sState.dy := fSim_Dy_Fix * pMark^.nId;
END_IF


// if marks are inverted (flipped along x-axis), the correction is inverted
IF NOT pMark^.bInvertedX THEN  pMark^.sState.dy := -1*pMark^.sState.dy; END_IF

// check position qualitiy
pMark^.sState.bInArea := FC_COMPARE_RANGE_PERCENT( 
                                       fI_ValueSet := (pMark^.fHeight / 2)
                                     , fI_ValueActual  := (pMark^.fHeight / 2) + pMark^.sState.dy
                                     , fI_RangePercent := nC_AreaMarkSensorOk);

                                     
setupMark := pMark^.sState.bSet;
END_METHOD

METHOD PRIVATE SheetStart
VAR_INPUT
  pMark : POINTER TO ST_MarkDefinition;
END_VAR
VAR
  sMarkBackup : ST_MarkDefinition;
END_VAR
_nX0 := pMark^.sState.nPosXReal - F_MeterToSubPixel(fPosMeter:=pMark^.fPosX, fResoSubPx:=_fResolution);
_bStartTrig := TRUE;
_fImageLengthEffective := _fImageLength;
bDetectionRunning := TRUE;
bNoStartMarkDetected := FALSE;
bInvalidRepeatLength := FALSE;
nInvalidSignalDetectedPerRepeat := 0;
nInvalidMarkDetectedPerRepeat := 0;

// (force) terminate a sheet/repeat
IF bSheetActive THEN 
  IF _bVerbose THEN LogInfo(F_Concat2('Terminate sheet/repeat with new Start Mark', '')); END_IF
  sMarkBackup := pMark^;   // push 
  SheetStop(nNewX0:=_nX0);
  pMark^:= sMarkBackup;    // pop
END_IF

IF _bVerbose THEN LogInfo(F_Concat2('SheetStart at X0=', TO_STRING(_nX0))); END_IF

// save (start) mark
_pFbMarkDefinition^.saveMark(pMark:=pMark);
SaveToMarkHistory(pMark:=pMarkSearch);    // Save to mark history

// trigger camera
IF _iActiveCam<>0 THEN _iActiveCam.CamTrigger(bOk:=TRUE, nPos:=_nX0, nPosDeviation:=0, nX0:=_nX0); END_IF

// save for supervision
nPosRepeatSupervision := _nX0;

bSheetActive := TRUE;
END_METHOD

METHOD PRIVATE SheetStop
VAR_INPUT
  nNewX0 : DINT;   // new detected X0
END_VAR
VAR_INST
  fSubstrateRealDiff : LREAL;   // [m]
  nSubstrareRealDiff : DINT;    // [SubPx]
END_VAR
VAR
  i : UDINT;
  pLastMark : POINTER TO ST_MarkDefinition;
  fD : LREAL;
  fSLen : LREAL;
  nDetectedX0 : DINT;
END_VAR
// - terminate
IF _bVerbose THEN LogInfo(F_Concat2('SheetStop()', '')); END_IF

fSLen := _fImageLength;  // (default) original length

// calculate effective sheet length
nDetectedX0 := getLastX0();   // get sampled X0
IF nNewX0 <> 0 AND nDetectedX0 <> 0 THEN
  // real diff between two starts
  fD := F_SubPixelToMeter(lPosSubPx:=nNewX0 - nDetectedX0, fResSubPx:=_fResolution);
  IF fD < (_fImageLength * fC_MaxSubstrateFactor) THEN
    fSLen := fD;
  END_IF 
ELSIF nNewX0 = 0 AND _pFbMarkDefinition^.nMarksDetected > 1 THEN
  // calculate based on last detected mark (a strech factor)
  pLastMark:= _pFbMarkDefinition^.getMark(nIdx:=0);     // get last available mark
  fD := getMarkDistanceEffective(pMark:=pLastMark); 
  fSLen := (pLastMark^.fPosX/SEL(fD<>0, pLastMark^.fPosX, fD)) * _fImageLength; // estimate real length with last mark
END_IF
_fImageLengthEffective := fSLen;
fSubstrateRealDiff := _fImageLengthEffective - _fImageLength;
nSubstrareRealDiff := (nNewX0 - nDetectedX0) - F_MeterToSubPixel(fPosMeter:=_fImageLength, fResoSubPx:=_fResolution);

// debug history
FOR i:=0 TO nC_HistorySize-1 DO sRepeatHistory[i].bSelected := FALSE; END_FOR   // clear selection
nRepeatCt := (nRepeatCt + 1) MOD nC_HistorySize;
sRepeatHistory[nRepeatCt].bSelected       := TRUE;
sRepeatHistory[nRepeatCt].nIndex          := nRepeatCt+1;
sRepeatHistory[nRepeatCt].nX0             := nDetectedX0;
sRepeatHistory[nRepeatCt].fLen            := _fImageLength * 1000;
sRepeatHistory[nRepeatCt].fLenEffective   := _fImageLengthEffective * 1000;
sRepeatHistory[nRepeatCt].fLenDiff        := (fSubstrateRealDiff) * 1000;
sRepeatHistory[nRepeatCt].bLenNotInRange  := bInvalidRepeatLength;
sRepeatHistory[nRepeatCt].bInvalidIngoredMarks := nInvalidMarkDetectedPerRepeat > 0;
sRepeatHistory[nRepeatCt].bMissingMarks   := nInvalidSignalDetectedPerRepeat > 0;


IF _iActiveCam<>0 THEN _iActiveCam.CamTriggerDone(); END_IF 
_pFbMarkDefinition^.ResetMarkStates();

bSheetActive := FALSE;
END_METHOD

METHOD PRIVATE SimMarks : BOOL
VAR_INPUT
  pMark : POINTER TO ST_MarkDefinition;
END_VAR
VAR_OUTPUT
  bStartMark : BOOL;
END_VAR
VAR_INST
  bMarkOn : BOOL;
  nMarkStarted : DINT;
  fStartMarkOffset : LREAL;
  rand : DRAND;
  rlrand : LREAL;
  l : LREAL;
  rf_ManuTrigger : RF_TRIG;
END_VAR
IF pMark = 0 THEN RETURN; END_IF

// when sim enabled AND auto-trigger then create a StartMark after every sheet/repeat length
//  then generate every following intermediate mark with a given length
rf_ManuTrigger(CLK:=bManualTrigger);
IF rf_ManuTrigger.RT THEN
  setupMark(
    pMark:=pMark,
    nDetectedPos:=nCurrentPos,
    fRealMarkLength:=F_MeterToSubPixelReal(fPosMeter:=pMark^.fSqLength + (pMark^.fTrLength/2), fResoSubPx:=_fResolution),
    bMissed:=FALSE
  );
  If pMark^.nId = 1 THEN bStartMark := TRUE; END_IF
  SimMarks := TRUE;
  RETURN;
END_IF


IF NOT bMarkOn THEN  // start new mark
  // create rising edge
  IF pMark^.nId = 1 THEN
    // wait for next StartPosition
    IF F_SubPixelToMeter(lPosSubPx:=ABS(nCurrentPos - nLastGeneratedStartMarkPosition), fResSubPx:=_fResolution) >= _fImageLength + _fSubstrateGap THEN
      nLastGeneratedStartMarkPosition := nCurrentPos;      // save start mark pos
      fStartMarkOffset := pMark^.fPosX;   // save start mark displacement from X0
      pMark^.sState.nPosXReal := nCurrentPos;  // save rising edge
      nMarkStarted := nCurrentPos;
      l := F_MeterToSubPixelReal(fPosMeter:=pMark^.fSqLength + (pMark^.fTrLength/2), fResoSubPx:=_fResolution); // mark length
      bMarkOn := TRUE;
    END_IF
	ELSE
    // wait for next mark position
    IF F_SubPixelToMeter(lPosSubPx:=ABS(nCurrentPos - nLastGeneratedStartMarkPosition), fResSubPx:=_fResolution) >= pMark^.fPosX - fStartMarkOffset THEN
      pMark^.sState.nPosXReal := nCurrentPos;  // save rising edge
      nMarkStarted := nCurrentPos;
      l := F_MeterToSubPixelReal(fPosMeter:=pMark^.fSqLength + (pMark^.fTrLength/2), fResoSubPx:=_fResolution); // mark length
      bMarkOn := TRUE;
		END_IF
  END_IF
  
ELSE
  // create falling edge
  IF (nCurrentPos - nMarkStarted) > l THEN
    rand(Seed:=13, Num=>rlrand);  // TODO: find a right scale 
    setupMark(
      pMark:=pMark,
      nDetectedPos:=nMarkStarted,
      fRealMarkLength:=F_SubPixelToMeter(lPosSubPx:=nCurrentPos - nMarkStarted, fResSubPx:=_fResolution),
      bMissed:=FALSE
    );
    bMarkOn := FALSE;
    If pMark^.nId = 1 THEN bStartMark := TRUE; END_IF
    SimMarks := TRUE;    // mark done
  END_IF
END_IF
END_METHOD

// simulate marks with sensor simulation
METHOD PRIVATE SimSensor
VAR_INPUT
END_VAR
VAR_OUTPUT
  bSensorSimulationSignal : BOOL;
  tSensorRising           : T_DCTIME64;
  tSensorFalling          : T_DCTIME64;
END_VAR
VAR
  fDistToLastStart : LREAL;
END_VAR
VAR_INST
  nNextMarkId : DINT;     // internal selection of marks
  bMarkOn : BOOL;         // sensor is on
  pMark : POINTER TO ST_MarkDefinition;  
  nPosMarkStarted : DINT;
  fStartMarkOffset : LREAL;
  SimMarkLength : LREAL;
  tRising, tFalling : T_DCTIME64;
END_VAR
IF _pFbMarkDefinition = 0 THEN RETURN; END_IF
IF nNextMarkId = 0 THEN nNextMarkId := 1; END_IF   // start with 1 always

IF NOT bMarkOn THEN  // start new mark

  pMark := _pFbMarkDefinition^.getMark(nIdx:=nNextMarkId);  // get theoretical mark configuration
  IF pMark <> 0 THEN
    // create rising edge
    IF pMark^.nId = 1 THEN
      // wait for next StartPosition
      fDistToLastStart := F_SubPixelToMeter(lPosSubPx:=ABS(nCurrentPos - nLastGeneratedStartMarkPosition), fResSubPx:=_fResolution); 
      IF fDistToLastStart >= _fImageLength + _fSubstrateGap THEN
        
        nPosMarkStarted := nCurrentPos;
        SimMarkLength := F_MeterToSubPixelReal(fPosMeter:=pMark^.fSqLength + (pMark^.fTrLength/2), fResoSubPx:=_fResolution); // mark length default
        
        nLastGeneratedStartMarkPosition := nCurrentPos;      // save start mark pos
        fStartMarkOffset := pMark^.fPosX;                    // save start mark displacement from X0
        tRising := tNowDc;
        bMarkOn := TRUE;
      END_IF
    ELSE
      // wait for next intermediate mark position
      fDistToLastStart := F_SubPixelToMeter(lPosSubPx:=ABS(nCurrentPos - nLastGeneratedStartMarkPosition), fResSubPx:=_fResolution);
      IF fDistToLastStart >= pMark^.fPosX - fStartMarkOffset THEN
        
        nPosMarkStarted := nCurrentPos;
        SimMarkLength := F_MeterToSubPixelReal(fPosMeter:=pMark^.fSqLength + (pMark^.fTrLength/2), fResoSubPx:=_fResolution); // mark length
        tRising := tNowDc;
        bMarkOn := TRUE;
      END_IF
    END_IF

  END_IF  
ELSE
  // create falling edge
  IF (nCurrentPos - nPosMarkStarted) >= SimMarkLength THEN
    tFalling := tNowDc;
    bMarkOn := FALSE;
    nNextMarkId := SEL(nNextMarkId = TO_DINT(_pFbMarkDefinition^.nMarks), nNextMarkId+1, 1);
  END_IF
END_IF

bSensorSimulationSignal := bMarkOn;
tSensorRising := tRising;
tSensorFalling := tFalling;
END_METHOD

METHOD strMark : T_MaxString
VAR_INPUT
  pMark : POINTER TO ST_MarkDefinition;
END_VAR
VAR_INST
  fbStrFormat : FB_FormatString;
END_VAR
VAR
  IdFormatted : STRING;
END_VAR
fbStrFormat(sFormat:='%.2d', arg1:=F_DINT(pMark^.nId), sOut=>IdFormatted);
strMark := F_Concat6(
  F_Concat2('Id:',   IdFormatted),
  F_Concat2(' Set:', SEL(pMark^.sState.bSet,'0','1')),
  F_Concat2(' posX:', LREAL_TO_FMTSTR( pMark^.fPosX, 5, TRUE )),
  F_Concat2(' posY:', LREAL_TO_FMTSTR( pMark^.fPosY, 5, TRUE )),
  F_Concat2(' dx:', LREAL_TO_FMTSTR( pMark^.sState.dx, 5, TRUE )),
  F_Concat2(' dy:', LREAL_TO_FMTSTR( pMark^.sState.dy, 5, TRUE )),
);
END_METHOD

END_FUNCTION_BLOCK

// ---- POUs/Print/Camera/Obsolete/FB_CAMERA_TRIGGER.TcPOU
FUNCTION_BLOCK FB_CAMERA_TRIGGER
(*************************************************************************************************)
(*  FILENAME:    FB_CAMERA_TRIGGER.EXP                                                           *)
(*  PROJECT:     CALMAR PUPLC                                                                    *)
(*  COPYRIGHT:   All rights reserved (c) Wifag//Polytype, Fribourg/Switzerland (2016)            *)
(*  ENVIRONMENT: TwinCAT PLC                                                                     *)
(*  VERSION:     <version>                                                                       *)
(*************************************************************************************************)
(*  DESCRIPTION:                                                                   <description> *)
(*    Generate timestamp trigger output based on timestamp sensor input. Two variants            *)
(*    exist, a timebased approach where the trigger time is calculated at the time the sensor    *)
(*    event occurs, and a second approach where the sensor event time is translated to a sensor  *)
(*    event position, and a trigger is generated when the calculated trigger position has almost *)
(*    been reached. The second approach has the advantage that is is less susceptible to speed   *)
(*    variations.                                                                                *)
(*                                                                                </description> *)
(*************************************************************************************************)

{library public}
VAR_INPUT
  (*From EL1252*)
  bI_Sensor_State                 : BOOL;            (*Sensor signal*)
  tI_Sensor_TimeStampPos          : T_DCTIME64;      (*Sensor last detection timestamp*)

  (*System signals*)
  iI_CurrentPos                   : DINT;            (*current position in Pulses/Subpixels*)
  fI_ConveyorSpeed                : REAL;            (*actual speed of conveyor in [m/s]*)
  fI_SubstrateLength              : REAL;            (*length of substrate in [m]*)
  bI_Reset                        : BOOL := FALSE;   (*reset this fb*)
  fI_TriggerDistance              : REAL;            (*Distance between Sensor and Trigger [m]*)
  bI_ManualTeachTrigger           : BOOL;            (*Generate teach trigger*)
  bI_ManualTrigger                : BOOL;            (*Generate test trigger*)

  (*configuration*)
  iI_Resolution                   : INT := 1;        (*Printhead Resolution [e.g. 600] x Subpixel Resolution [e.g. 32]*)
  bI_UsePositionTrigger           : BOOL;            (*FALSE: Calculate time with speed and position distance@sensor evont*)
                                                     (*TRUE:   Calculate sensor event position, launch trigger based on position*)
  fL_TriggerLength                : LREAL := 0.1;    (*Length of trigger signal in ms, min. 3 bus cycles*)
END_VAR

VAR_OUTPUT
  (*Link to EL2252*)
  tO_Trigger_StartTime            : T_DCTIME64;      (*Link to EL2252 StartTime*)
  bO_Trigger                      : BOOL;            (*Link to EL2252 Output*)
  cO_Activate                     : BYTE;            (*Link to EL2252 Activate*)
  bO_Active                       : BOOL;            (*True when Trigger generation started*)
END_VAR

(*{library private}*)
VAR
  bL_SpeedValid                   : BOOL;
  bL_InhibitTrigger               : BOOL;            (*inhibit trigger signals, TRUE=inhibit*)
  bL_ReleaseInhibitTrigger        : BOOL;            (*condition to release inhibit trigger*)

  cL_State                        : BYTE;            (*State*)
  tL_Sensor_TimeStamp             : T_DCTIME64;      (*Sensor last detection timestamp*)
  tL_CurrentTime                  : T_DCTIME64;      (*Current system time*)
  tL_Trigger_EventTime            : T_DCTIME64;      (*Trigger event timestamp*)

  fL_DeltaDistance                : LREAL;           (*Distance that the substrate moved between the detection and the treatment of the information [m]*)
  iL_StartPos                     : DINT;            (*Sensor start position [SubPx]*)
  iL_SubstrateLength              : DINT;            (*Substrate length in pulse [SubPx]*)

  tL_CurrentTimeStamp             : T_DCTIME64;      (* Get Current Timestamp *)
  tL_LastTimeStamp                : T_DCTIME64;      (* Get Current Timestamp *)
  fL_DeltaTimeStamp               : LREAL;           (* Get Current Timestamp *)

  fL_RemDist                      : LREAL;           (*Remaining distance until trigger occurs [m]*)
  fL_PreTriggerPosition           : LREAL;           (*Margin between effective trigger position and generation of timestamp*)

  fb_FTrig_ManualTeach            : F_TRIG;          (*FTrig for teach to release inhibit*)
END_VAR

VAR CONSTANT
  fC_MIN_CONVEYOR_SPEED           : REAL := 0.05;
  fC_PRETRIGFACTOR                : REAL := 3.0;

  (*State*)
  cL_IDLE                         : BYTE := 0;       (*Idle state, no trigger active*)
  cL_SENSOREVENT                  : BYTE := 1;       (*Sensor started trigger generation*)
  cL_WAITALMOSTSTART              : BYTE := 2;       (*Wait timestamp calculation critera*)
  cL_WAITSTART                    : BYTE := 3;       (*Wait for trigger generation critera*)
  cL_TRIGACTIVE                   : BYTE := 4;       (*Trigger set*)
  cL_WAITSTOP                     : BYTE := 5;       (*Trigger reset*)

  (*EL2252 Command*)
  cL_INACTIVE                     : BYTE := 0;
  cL_ACTIVE                       : BYTE := 3;
END_VAR

IF bI_Reset THEN
  cL_State          := cL_IDLE;
	bL_InhibitTrigger := FALSE;
END_IF;

(*zero divisions*)
IF iI_Resolution = 0 THEN RETURN; END_IF;

(*General calculations*)
bL_SpeedValid     := fI_ConveyorSpeed > fC_MIN_CONVEYOR_SPEED;
tL_CurrentTime    := F_GetCurDcTaskTime64();
fL_DeltaTimeStamp := (ULINT_TO_LREAL(tL_CurrentTime) - ULINT_TO_LREAL(tL_LastTimeStamp)) * 1E-9;
tL_LastTimeStamp  := tL_CurrentTime;

(*Added 10 mm margin for substrate length in case of print quality strips at the end of sheet in case of start with edge*)
iL_SubstrateLength := FC_LREAL_TO_DINT((fI_SubstrateLength + 0.01) * (1 / (0.0254 / iI_Resolution)));


(*State Machine ----------------------------------------------------------------*)
CASE cL_State OF
  cL_IDLE:     (*Not started*)
    IF bL_SpeedValid AND bI_Sensor_State AND NOT bL_InhibitTrigger THEN      (*Start launched*)
      cL_State            := cL_SENSOREVENT;
      tL_Sensor_TimeStamp := tI_Sensor_TimeStampPos;
    ELSIF     (   (bL_SpeedValid AND bI_ManualTrigger)
               OR bI_ManualTeachTrigger
              )
          AND NOT bL_InhibitTrigger
    THEN  (*Manual start launched*)
      cL_State            := cL_SENSOREVENT;
      tL_Sensor_TimeStamp := tL_CurrentTime;
    ELSE
      cL_State     := cL_IDLE;
    END_IF;

    cO_Activate    := cL_INACTIVE;
    bO_Trigger     := FALSE;
    bO_Active      := FALSE;

  cL_SENSOREVENT:     (*Not started*)
    IF bI_ManualTeachTrigger THEN
      cL_State             := cL_WAITSTART;

    (*tL_Trigger_EventTime := UInt64Add64(ULINT_TO_ULARGE(tL_Sensor_TimeStamp), LREAL_TO_UINT64(100 * 1E6));  (*delay 100ms*)*)
      tL_Trigger_EventTime := (tL_Sensor_TimeStamp + LREAL_TO_ULINT(100 * 1E6));  (*delay 100ms*)
      iL_StartPos          := iI_CurrentPos;

      cO_Activate          := cL_INACTIVE;
    ELSE
      IF bI_UsePositionTrigger THEN
        cL_State             := cL_WAITALMOSTSTART;

        (*Distance in pulses that the substrate has traveled between the sensor detection and the PLC treatment*)
        fL_DeltaDistance     := UINT64_TO_LREAL(UInt64Sub64(ULINT_TO_ULARGE(tL_CurrentTime), ULINT_TO_ULARGE(tL_Sensor_TimeStamp))) * 1E-9 * fI_ConveyorSpeed;
        (*Position where the sheet has been detected*)
        iL_StartPos          := iI_CurrentPos - FC_LREAL_TO_DINT(fL_DeltaDistance * (1 / (0.0254 / INT_TO_REAL(iI_Resolution))));
      ELSE
        cL_State             := cL_WAITSTART;

